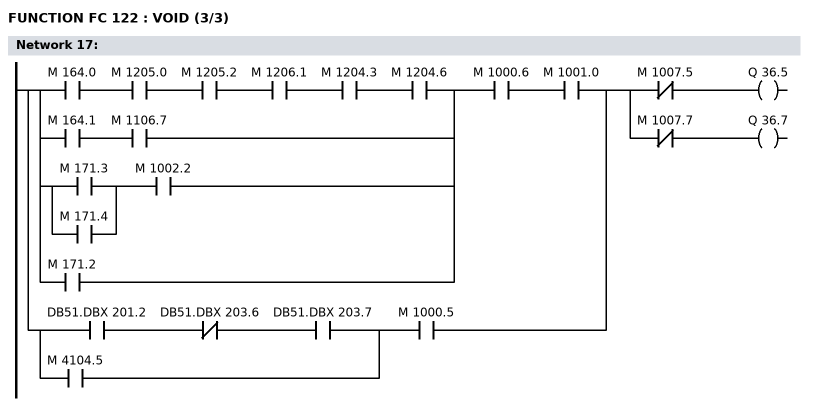

      A(    ;
      A     M    164.0;
      A     M   1205.0;
      A     M   1205.2;
      A     M   1206.1;
      A     M   1204.3;
      A     M   1204.6;
      O     ;
      A     M    164.1;
      A     M   1106.7;
      O     ;
      A(    ;
      O     M    171.3;
      O     M    171.4;
      )     ;
      A     M   1002.2;
      O     M    171.2;
      )     ;
      A     M   1000.6;
      A     M   1001.0;
      O     ;
      A(    ;
      A     DB51.DBX  201.2;
      AN    DB51.DBX  203.6;
      A     DB51.DBX  203.7;
      O     M   4104.5;
      )     ;
      A     M   1000.5;
      =     L      0.0;
      A     L      0.0;
      AN    M   1007.5;
      =     Q     36.5;
      A     L      0.0;
      AN    M   1007.7;
      =     Q     36.7;
END_FUNCTION

FUNCTION_BLOCK FB 123
TITLE =
VERSION : 0.1


VAR
  S706_LM_DC_PIN : FB 424;
  S706_LM_DC_1ST_CLAMP1 : FB 424;
  S706_LM_DC_1ST_CLAMP2 : FB 424;
  S706_LM_DC_1ST_CLAMP3 : FB 424;
  S706_LM_DC_1ST_CLAMP4 : FB 424;
  S706_LM_DC_2ND_CLAMP1 : FB 424;
  S706_LM_DC_2ND_CLAMP2 : FB 424;
  S706_LM_DC_2ND_CLAMP3 : FB 424;
  S706_LM_DC_2ND_CLAMP4 : FB 424;
  S706_LM_DC_2ND_CLAMP5 : FB 424;
  S706_LM_DC_STK_PIN : FB 424;
  S706_LM_DC_OTR_CLAMP : FB 424;
  S706_LM_DC_ASSY_CLAMP : FB 424;
  S706_LM_DC_FF_PIN : FB 424;
  S706_LM_DC_FF_CLAMP : FB 424;
  S706_LM_DC_2ND_CLAMP6 : FB 424;
  S706_LM_DC_2ND_CLAMP7 : FB 424;
  S706_LM_DC_1ST_CLAMP5 : FB 424;
END_VAR
BEGIN
NETWORK
TITLE =
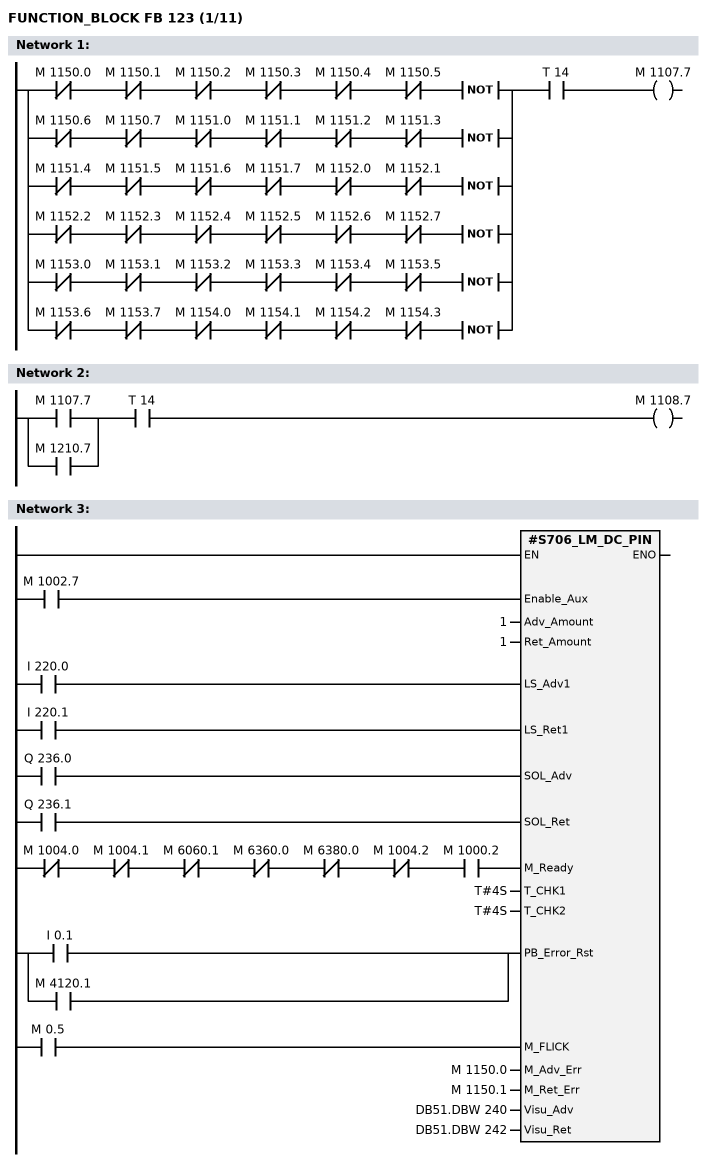

      A(    ;
      AN    M   1150.0;
      AN    M   1150.1;
      AN    M   1150.2;
      AN    M   1150.3;
      AN    M   1150.4;
      AN    M   1150.5;
      NOT   ;
      O(    ;
      AN    M   1150.6;
      AN    M   1150.7;
      AN    M   1151.0;
      AN    M   1151.1;
      AN    M   1151.2;
      AN    M   1151.3;
      NOT   ;
      )     ;
      O(    ;
      AN    M   1151.4;
      AN    M   1151.5;
      AN    M   1151.6;
      AN    M   1151.7;
      AN    M   1152.0;
      AN    M   1152.1;
      NOT   ;
      )     ;
      O(    ;
      AN    M   1152.2;
      AN    M   1152.3;
      AN    M   1152.4;
      AN    M   1152.5;
      AN    M   1152.6;
      AN    M   1152.7;
      NOT   ;
      )     ;
      O(    ;
      AN    M   1153.0;
      AN    M   1153.1;
      AN    M   1153.2;
      AN    M   1153.3;
      AN    M   1153.4;
      AN    M   1153.5;
      NOT   ;
      )     ;
      O(    ;
      AN    M   1153.6;
      AN    M   1153.7;
      AN    M   1154.0;
      AN    M   1154.1;
      AN    M   1154.2;
      AN    M   1154.3;
      NOT   ;
      )     ;
      )     ;
      A     T     14;
      =     M   1107.7;
NETWORK
TITLE =

      A(    ;
      O     M   1107.7;
      O     M   1210.7;
      )     ;
      A     T     14;
      =     M   1108.7;
NETWORK
TITLE =

      A     M   1002.7;
      =     L      0.0;
      BLD   103;
      A     I    220.0;
      =     L      0.1;
      BLD   103;
      A     I    220.1;
      =     L      0.2;
      BLD   103;
      A     Q    236.0;
      =     L      1.1;
      BLD   103;
      A     Q    236.1;
      =     L      1.2;
      BLD   103;
      AN    M   1004.0;
      AN    M   1004.1;
      AN    M   6060.1;
      AN    M   6360.0;
      AN    M   6380.0;
      AN    M   1004.2;
      A     M   1000.2;
      =     L      1.3;
      BLD   103;
      A(    ;
      O     I      0.1;
      O     M   4120.1;
      )     ;
      =     L      1.5;
      BLD   103;
      A     M      0.5;
      =     L      1.6;
      BLD   103;
      CALL #S706_LM_DC_PIN (
           Enable_Aux               := L      0.0,
           Adv_Amount               := 1,
           Ret_Amount               := 1,
           LS_Adv1                  := L      0.1,
           LS_Ret1                  := L      0.2,
           SOL_Adv                  := L      1.1,
           SOL_Ret                  := L      1.2,
           M_Ready                  := L      1.3,
           T_CHK1                   := T#4S,
           T_CHK2                   := T#4S,
           PB_Error_Rst             := L      1.5,
           M_FLICK                  := L      1.6,
           M_Adv_Err                := M   1150.0,
           M_Ret_Err                := M   1150.1,
           Visu_Adv                 := DB51.DBW  240,
           Visu_Ret                 := DB51.DBW  242);
      NOP   0;
NETWORK
TITLE =
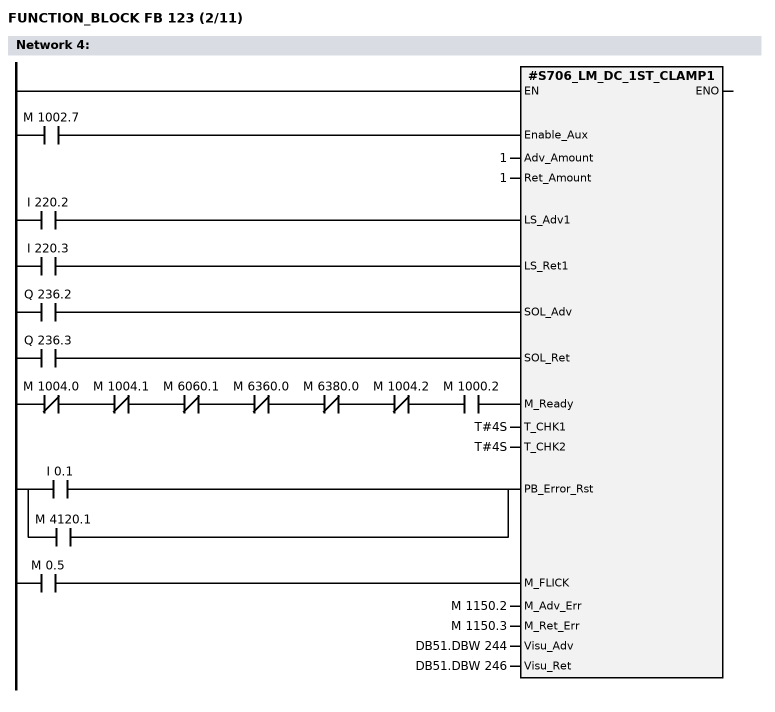

      A     M   1002.7;
      =     L      0.0;
      BLD   103;
      A     I    220.2;
      =     L      0.1;
      BLD   103;
      A     I    220.3;
      =     L      0.2;
      BLD   103;
      A     Q    236.2;
      =     L      1.1;
      BLD   103;
      A     Q    236.3;
      =     L      1.2;
      BLD   103;
      AN    M   1004.0;
      AN    M   1004.1;
      AN    M   6060.1;
      AN    M   6360.0;
      AN    M   6380.0;
      AN    M   1004.2;
      A     M   1000.2;
      =     L      1.3;
      BLD   103;
      A(    ;
      O     I      0.1;
      O     M   4120.1;
      )     ;
      =     L      1.5;
      BLD   103;
      A     M      0.5;
      =     L      1.6;
      BLD   103;
      CALL #S706_LM_DC_1ST_CLAMP1 (
           Enable_Aux               := L      0.0,
           Adv_Amount               := 1,
           Ret_Amount               := 1,
           LS_Adv1                  := L      0.1,
           LS_Ret1                  := L      0.2,
           SOL_Adv                  := L      1.1,
           SOL_Ret                  := L      1.2,
           M_Ready                  := L      1.3,
           T_CHK1                   := T#4S,
           T_CHK2                   := T#4S,
           PB_Error_Rst             := L      1.5,
           M_FLICK                  := L      1.6,
           M_Adv_Err                := M   1150.2,
           M_Ret_Err                := M   1150.3,
           Visu_Adv                 := DB51.DBW  244,
           Visu_Ret                 := DB51.DBW  246);
      NOP   0;
NETWORK
TITLE =
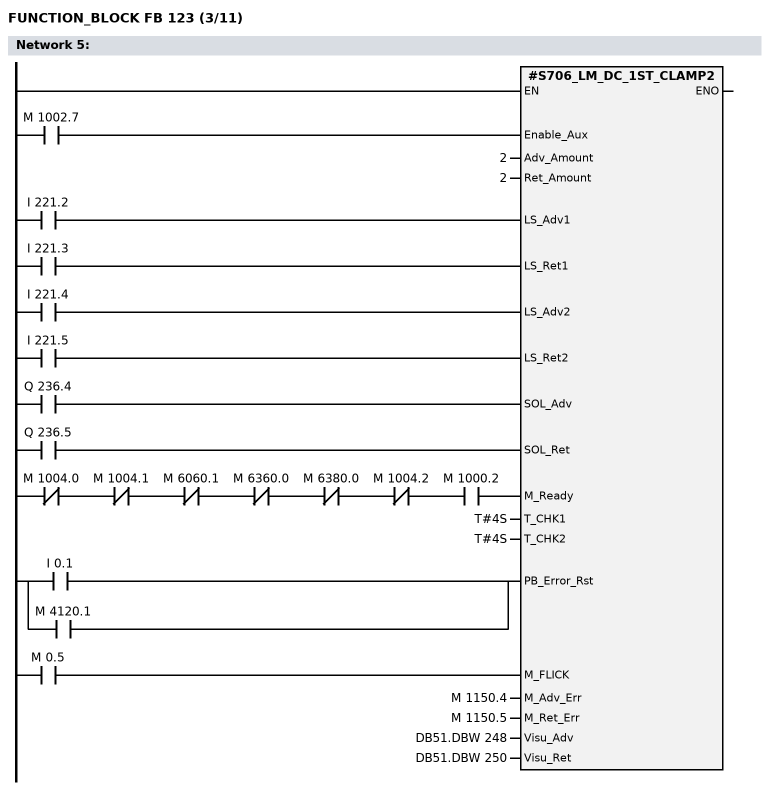

      A     M   1002.7;
      =     L      0.0;
      BLD   103;
      A     I    221.2;
      =     L      0.1;
      BLD   103;
      A     I    221.3;
      =     L      0.2;
      BLD   103;
      A     I    221.4;
      =     L      0.3;
      BLD   103;
      A     I    221.5;
      =     L      0.4;
      BLD   103;
      A     Q    236.4;
      =     L      1.1;
      BLD   103;
      A     Q    236.5;
      =     L      1.2;
      BLD   103;
      AN    M   1004.0;
      AN    M   1004.1;
      AN    M   6060.1;
      AN    M   6360.0;
      AN    M   6380.0;
      AN    M   1004.2;
      A     M   1000.2;
      =     L      1.3;
      BLD   103;
      A(    ;
      O     I      0.1;
      O     M   4120.1;
      )     ;
      =     L      1.5;
      BLD   103;
      A     M      0.5;
      =     L      1.6;
      BLD   103;
      CALL #S706_LM_DC_1ST_CLAMP2 (
           Enable_Aux               := L      0.0,
           Adv_Amount               := 2,
           Ret_Amount               := 2,
           LS_Adv1                  := L      0.1,
           LS_Ret1                  := L      0.2,
           LS_Adv2                  := L      0.3,
           LS_Ret2                  := L      0.4,
           SOL_Adv                  := L      1.1,
           SOL_Ret                  := L      1.2,
           M_Ready                  := L      1.3,
           T_CHK1                   := T#4S,
           T_CHK2                   := T#4S,
           PB_Error_Rst             := L      1.5,
           M_FLICK                  := L      1.6,
           M_Adv_Err                := M   1150.4,
           M_Ret_Err                := M   1150.5,
           Visu_Adv                 := DB51.DBW  248,
           Visu_Ret                 := DB51.DBW  250);
      NOP   0;
NETWORK
TITLE =
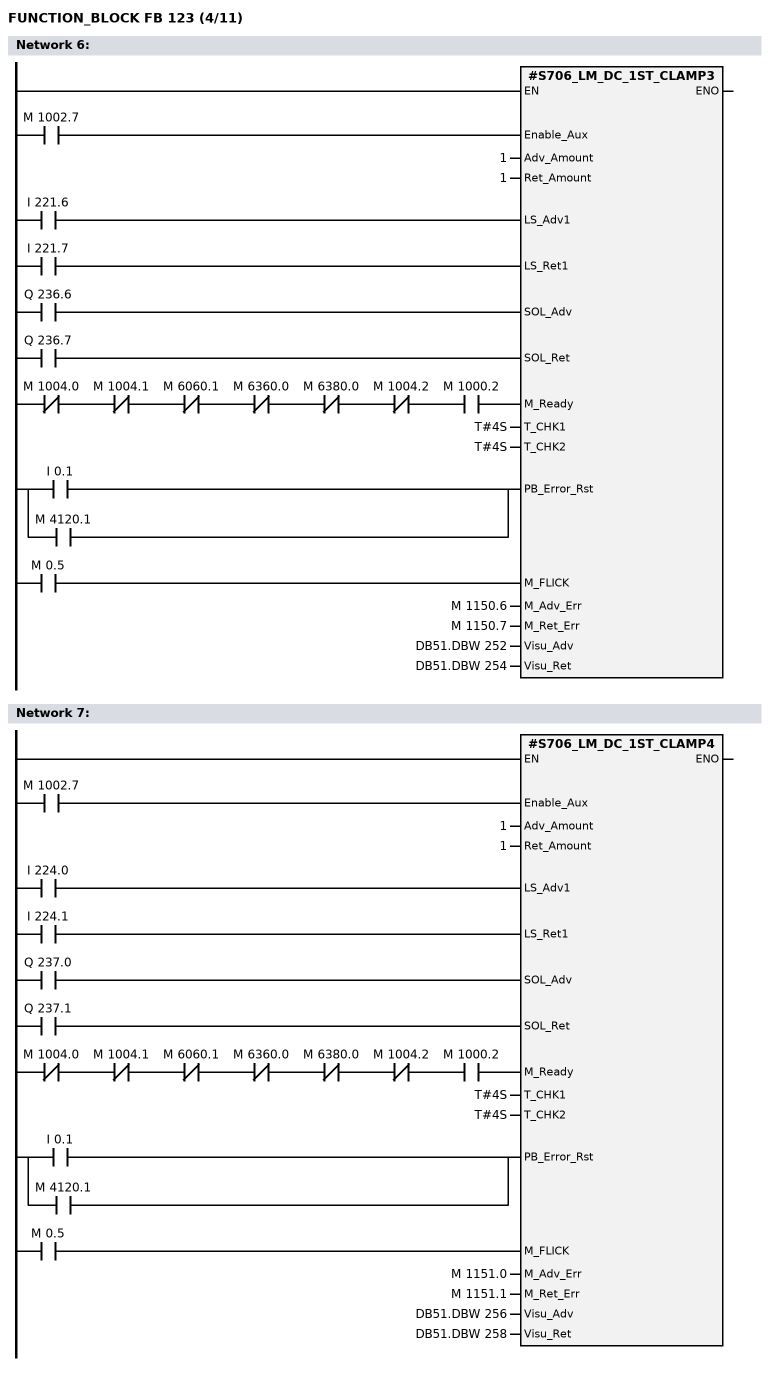

      A     M   1002.7;
      =     L      0.0;
      BLD   103;
      A     I    221.6;
      =     L      0.1;
      BLD   103;
      A     I    221.7;
      =     L      0.2;
      BLD   103;
      A     Q    236.6;
      =     L      1.1;
      BLD   103;
      A     Q    236.7;
      =     L      1.2;
      BLD   103;
      AN    M   1004.0;
      AN    M   1004.1;
      AN    M   6060.1;
      AN    M   6360.0;
      AN    M   6380.0;
      AN    M   1004.2;
      A     M   1000.2;
      =     L      1.3;
      BLD   103;
      A(    ;
      O     I      0.1;
      O     M   4120.1;
      )     ;
      =     L      1.5;
      BLD   103;
      A     M      0.5;
      =     L      1.6;
      BLD   103;
      CALL #S706_LM_DC_1ST_CLAMP3 (
           Enable_Aux               := L      0.0,
           Adv_Amount               := 1,
           Ret_Amount               := 1,
           LS_Adv1                  := L      0.1,
           LS_Ret1                  := L      0.2,
           SOL_Adv                  := L      1.1,
           SOL_Ret                  := L      1.2,
           M_Ready                  := L      1.3,
           T_CHK1                   := T#4S,
           T_CHK2                   := T#4S,
           PB_Error_Rst             := L      1.5,
           M_FLICK                  := L      1.6,
           M_Adv_Err                := M   1150.6,
           M_Ret_Err                := M   1150.7,
           Visu_Adv                 := DB51.DBW  252,
           Visu_Ret                 := DB51.DBW  254);
      NOP   0;
NETWORK
TITLE =

      A     M   1002.7;
      =     L      0.0;
      BLD   103;
      A     I    224.0;
      =     L      0.1;
      BLD   103;
      A     I    224.1;
      =     L      0.2;
      BLD   103;
      A     Q    237.0;
      =     L      1.1;
      BLD   103;
      A     Q    237.1;
      =     L      1.2;
      BLD   103;
      AN    M   1004.0;
      AN    M   1004.1;
      AN    M   6060.1;
      AN    M   6360.0;
      AN    M   6380.0;
      AN    M   1004.2;
      A     M   1000.2;
      =     L      1.3;
      BLD   103;
      A(    ;
      O     I      0.1;
      O     M   4120.1;
      )     ;
      =     L      1.5;
      BLD   103;
      A     M      0.5;
      =     L      1.6;
      BLD   103;
      CALL #S706_LM_DC_1ST_CLAMP4 (
           Enable_Aux               := L      0.0,
           Adv_Amount               := 1,
           Ret_Amount               := 1,
           LS_Adv1                  := L      0.1,
           LS_Ret1                  := L      0.2,
           SOL_Adv                  := L      1.1,
           SOL_Ret                  := L      1.2,
           M_Ready                  := L      1.3,
           T_CHK1                   := T#4S,
           T_CHK2                   := T#4S,
           PB_Error_Rst             := L      1.5,
           M_FLICK                  := L      1.6,
           M_Adv_Err                := M   1151.0,
           M_Ret_Err                := M   1151.1,
           Visu_Adv                 := DB51.DBW  256,
           Visu_Ret                 := DB51.DBW  258);
      NOP   0;
NETWORK
TITLE =
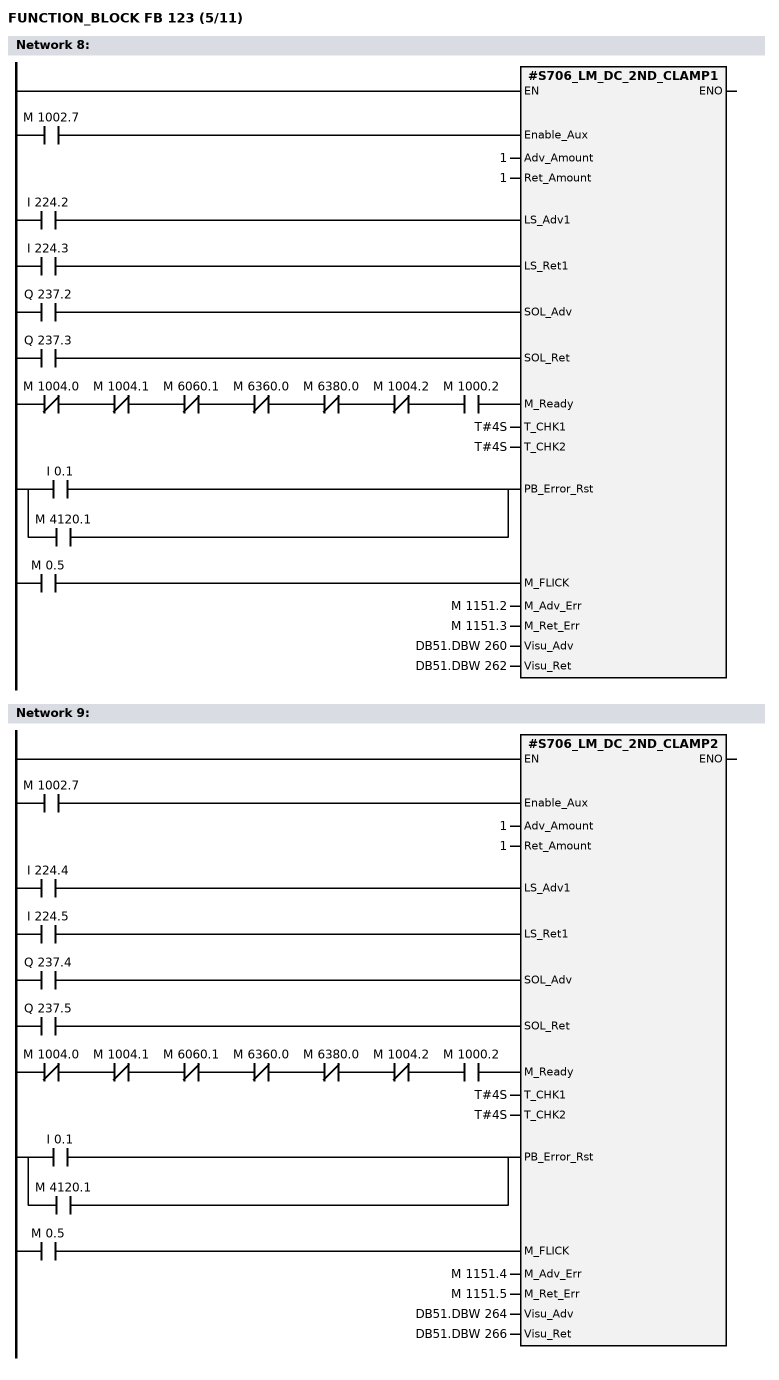

      A     M   1002.7;
      =     L      0.0;
      BLD   103;
      A     I    224.2;
      =     L      0.1;
      BLD   103;
      A     I    224.3;
      =     L      0.2;
      BLD   103;
      A     Q    237.2;
      =     L      1.1;
      BLD   103;
      A     Q    237.3;
      =     L      1.2;
      BLD   103;
      AN    M   1004.0;
      AN    M   1004.1;
      AN    M   6060.1;
      AN    M   6360.0;
      AN    M   6380.0;
      AN    M   1004.2;
      A     M   1000.2;
      =     L      1.3;
      BLD   103;
      A(    ;
      O     I      0.1;
      O     M   4120.1;
      )     ;
      =     L      1.5;
      BLD   103;
      A     M      0.5;
      =     L      1.6;
      BLD   103;
      CALL #S706_LM_DC_2ND_CLAMP1 (
           Enable_Aux               := L      0.0,
           Adv_Amount               := 1,
           Ret_Amount               := 1,
           LS_Adv1                  := L      0.1,
           LS_Ret1                  := L      0.2,
           SOL_Adv                  := L      1.1,
           SOL_Ret                  := L      1.2,
           M_Ready                  := L      1.3,
           T_CHK1                   := T#4S,
           T_CHK2                   := T#4S,
           PB_Error_Rst             := L      1.5,
           M_FLICK                  := L      1.6,
           M_Adv_Err                := M   1151.2,
           M_Ret_Err                := M   1151.3,
           Visu_Adv                 := DB51.DBW  260,
           Visu_Ret                 := DB51.DBW  262);
      NOP   0;
NETWORK
TITLE =

      A     M   1002.7;
      =     L      0.0;
      BLD   103;
      A     I    224.4;
      =     L      0.1;
      BLD   103;
      A     I    224.5;
      =     L      0.2;
      BLD   103;
      A     Q    237.4;
      =     L      1.1;
      BLD   103;
      A     Q    237.5;
      =     L      1.2;
      BLD   103;
      AN    M   1004.0;
      AN    M   1004.1;
      AN    M   6060.1;
      AN    M   6360.0;
      AN    M   6380.0;
      AN    M   1004.2;
      A     M   1000.2;
      =     L      1.3;
      BLD   103;
      A(    ;
      O     I      0.1;
      O     M   4120.1;
      )     ;
      =     L      1.5;
      BLD   103;
      A     M      0.5;
      =     L      1.6;
      BLD   103;
      CALL #S706_LM_DC_2ND_CLAMP2 (
           Enable_Aux               := L      0.0,
           Adv_Amount               := 1,
           Ret_Amount               := 1,
           LS_Adv1                  := L      0.1,
           LS_Ret1                  := L      0.2,
           SOL_Adv                  := L      1.1,
           SOL_Ret                  := L      1.2,
           M_Ready                  := L      1.3,
           T_CHK1                   := T#4S,
           T_CHK2                   := T#4S,
           PB_Error_Rst             := L      1.5,
           M_FLICK                  := L      1.6,
           M_Adv_Err                := M   1151.4,
           M_Ret_Err                := M   1151.5,
           Visu_Adv                 := DB51.DBW  264,
           Visu_Ret                 := DB51.DBW  266);
      NOP   0;
NETWORK
TITLE =
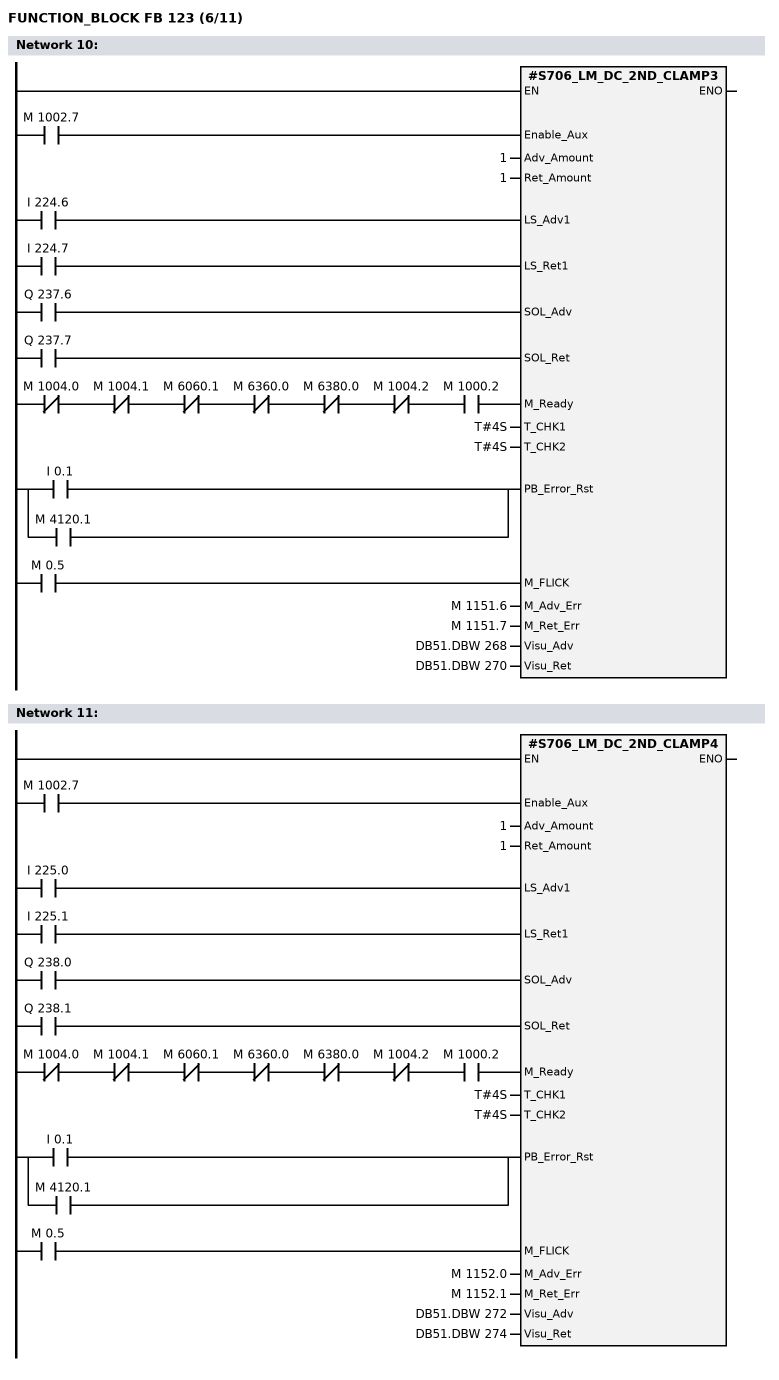

      A     M   1002.7;
      =     L      0.0;
      BLD   103;
      A     I    224.6;
      =     L      0.1;
      BLD   103;
      A     I    224.7;
      =     L      0.2;
      BLD   103;
      A     Q    237.6;
      =     L      1.1;
      BLD   103;
      A     Q    237.7;
      =     L      1.2;
      BLD   103;
      AN    M   1004.0;
      AN    M   1004.1;
      AN    M   6060.1;
      AN    M   6360.0;
      AN    M   6380.0;
      AN    M   1004.2;
      A     M   1000.2;
      =     L      1.3;
      BLD   103;
      A(    ;
      O     I      0.1;
      O     M   4120.1;
      )     ;
      =     L      1.5;
      BLD   103;
      A     M      0.5;
      =     L      1.6;
      BLD   103;
      CALL #S706_LM_DC_2ND_CLAMP3 (
           Enable_Aux               := L      0.0,
           Adv_Amount               := 1,
           Ret_Amount               := 1,
           LS_Adv1                  := L      0.1,
           LS_Ret1                  := L      0.2,
           SOL_Adv                  := L      1.1,
           SOL_Ret                  := L      1.2,
           M_Ready                  := L      1.3,
           T_CHK1                   := T#4S,
           T_CHK2                   := T#4S,
           PB_Error_Rst             := L      1.5,
           M_FLICK                  := L      1.6,
           M_Adv_Err                := M   1151.6,
           M_Ret_Err                := M   1151.7,
           Visu_Adv                 := DB51.DBW  268,
           Visu_Ret                 := DB51.DBW  270);
      NOP   0;
NETWORK
TITLE =

      A     M   1002.7;
      =     L      0.0;
      BLD   103;
      A     I    225.0;
      =     L      0.1;
      BLD   103;
      A     I    225.1;
      =     L      0.2;
      BLD   103;
      A     Q    238.0;
      =     L      1.1;
      BLD   103;
      A     Q    238.1;
      =     L      1.2;
      BLD   103;
      AN    M   1004.0;
      AN    M   1004.1;
      AN    M   6060.1;
      AN    M   6360.0;
      AN    M   6380.0;
      AN    M   1004.2;
      A     M   1000.2;
      =     L      1.3;
      BLD   103;
      A(    ;
      O     I      0.1;
      O     M   4120.1;
      )     ;
      =     L      1.5;
      BLD   103;
      A     M      0.5;
      =     L      1.6;
      BLD   103;
      CALL #S706_LM_DC_2ND_CLAMP4 (
           Enable_Aux               := L      0.0,
           Adv_Amount               := 1,
           Ret_Amount               := 1,
           LS_Adv1                  := L      0.1,
           LS_Ret1                  := L      0.2,
           SOL_Adv                  := L      1.1,
           SOL_Ret                  := L      1.2,
           M_Ready                  := L      1.3,
           T_CHK1                   := T#4S,
           T_CHK2                   := T#4S,
           PB_Error_Rst             := L      1.5,
           M_FLICK                  := L      1.6,
           M_Adv_Err                := M   1152.0,
           M_Ret_Err                := M   1152.1,
           Visu_Adv                 := DB51.DBW  272,
           Visu_Ret                 := DB51.DBW  274);
      NOP   0;
NETWORK
TITLE =
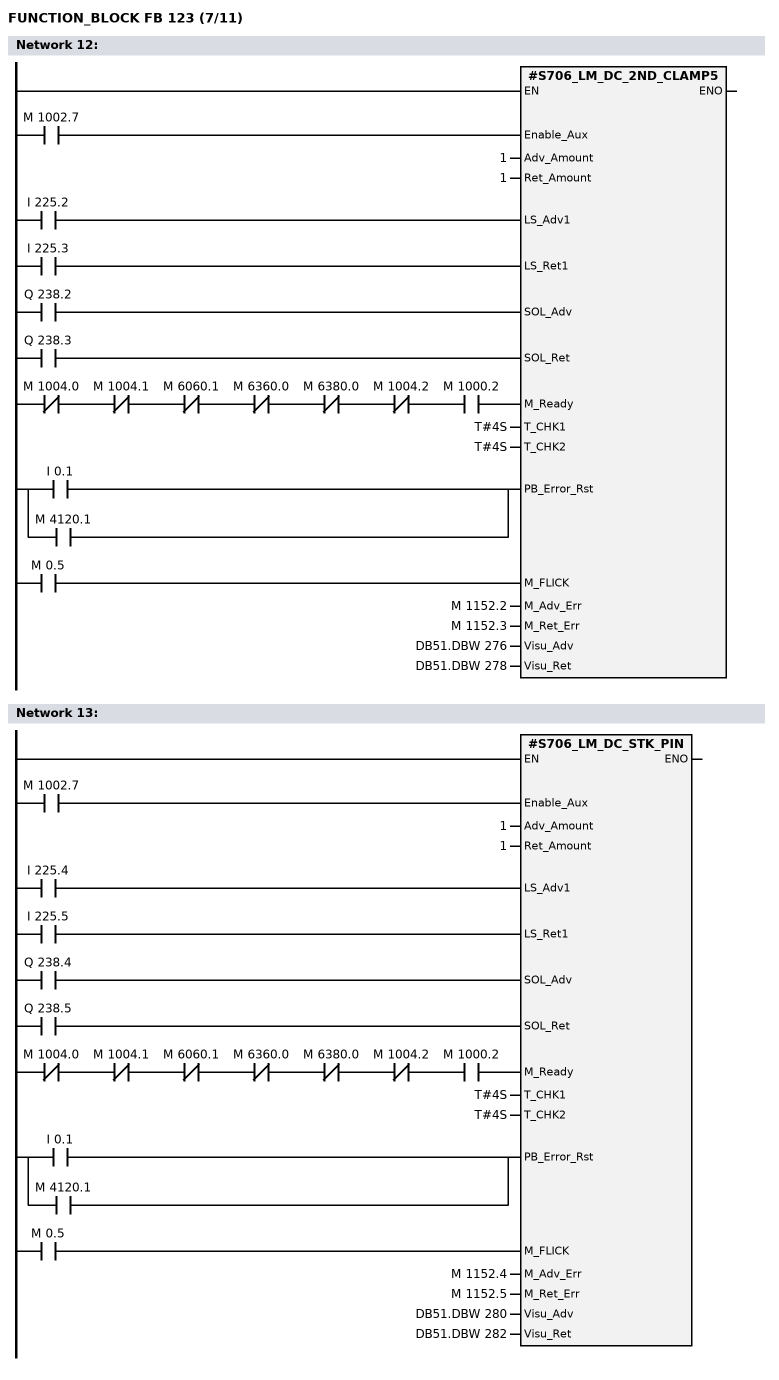

      A     M   1002.7;
      =     L      0.0;
      BLD   103;
      A     I    225.2;
      =     L      0.1;
      BLD   103;
      A     I    225.3;
      =     L      0.2;
      BLD   103;
      A     Q    238.2;
      =     L      1.1;
      BLD   103;
      A     Q    238.3;
      =     L      1.2;
      BLD   103;
      AN    M   1004.0;
      AN    M   1004.1;
      AN    M   6060.1;
      AN    M   6360.0;
      AN    M   6380.0;
      AN    M   1004.2;
      A     M   1000.2;
      =     L      1.3;
      BLD   103;
      A(    ;
      O     I      0.1;
      O     M   4120.1;
      )     ;
      =     L      1.5;
      BLD   103;
      A     M      0.5;
      =     L      1.6;
      BLD   103;
      CALL #S706_LM_DC_2ND_CLAMP5 (
           Enable_Aux               := L      0.0,
           Adv_Amount               := 1,
           Ret_Amount               := 1,
           LS_Adv1                  := L      0.1,
           LS_Ret1                  := L      0.2,
           SOL_Adv                  := L      1.1,
           SOL_Ret                  := L      1.2,
           M_Ready                  := L      1.3,
           T_CHK1                   := T#4S,
           T_CHK2                   := T#4S,
           PB_Error_Rst             := L      1.5,
           M_FLICK                  := L      1.6,
           M_Adv_Err                := M   1152.2,
           M_Ret_Err                := M   1152.3,
           Visu_Adv                 := DB51.DBW  276,
           Visu_Ret                 := DB51.DBW  278);
      NOP   0;
NETWORK
TITLE =

      A     M   1002.7;
      =     L      0.0;
      BLD   103;
      A     I    225.4;
      =     L      0.1;
      BLD   103;
      A     I    225.5;
      =     L      0.2;
      BLD   103;
      A     Q    238.4;
      =     L      1.1;
      BLD   103;
      A     Q    238.5;
      =     L      1.2;
      BLD   103;
      AN    M   1004.0;
      AN    M   1004.1;
      AN    M   6060.1;
      AN    M   6360.0;
      AN    M   6380.0;
      AN    M   1004.2;
      A     M   1000.2;
      =     L      1.3;
      BLD   103;
      A(    ;
      O     I      0.1;
      O     M   4120.1;
      )     ;
      =     L      1.5;
      BLD   103;
      A     M      0.5;
      =     L      1.6;
      BLD   103;
      CALL #S706_LM_DC_STK_PIN (
           Enable_Aux               := L      0.0,
           Adv_Amount               := 1,
           Ret_Amount               := 1,
           LS_Adv1                  := L      0.1,
           LS_Ret1                  := L      0.2,
           SOL_Adv                  := L      1.1,
           SOL_Ret                  := L      1.2,
           M_Ready                  := L      1.3,
           T_CHK1                   := T#4S,
           T_CHK2                   := T#4S,
           PB_Error_Rst             := L      1.5,
           M_FLICK                  := L      1.6,
           M_Adv_Err                := M   1152.4,
           M_Ret_Err                := M   1152.5,
           Visu_Adv                 := DB51.DBW  280,
           Visu_Ret                 := DB51.DBW  282);
      NOP   0;
NETWORK
TITLE =
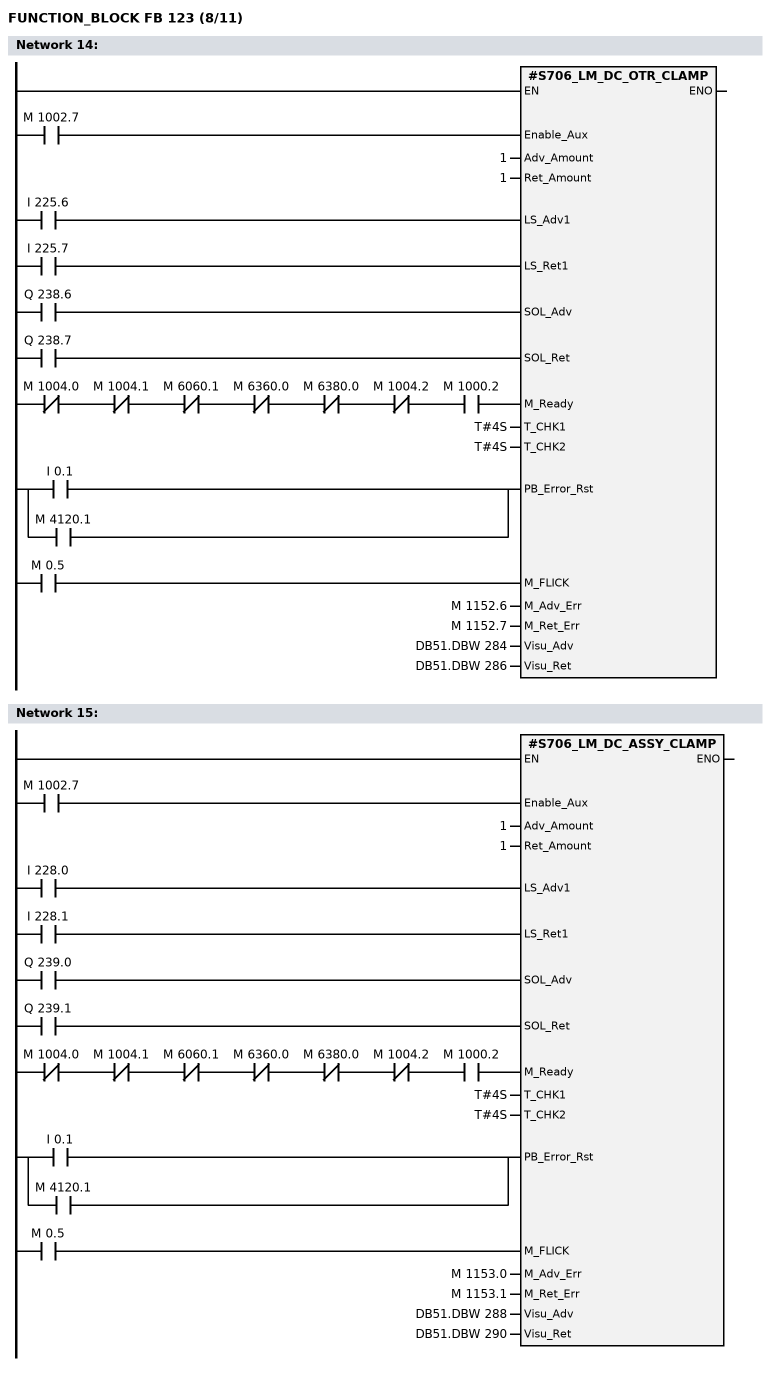

      A     M   1002.7;
      =     L      0.0;
      BLD   103;
      A     I    225.6;
      =     L      0.1;
      BLD   103;
      A     I    225.7;
      =     L      0.2;
      BLD   103;
      A     Q    238.6;
      =     L      1.1;
      BLD   103;
      A     Q    238.7;
      =     L      1.2;
      BLD   103;
      AN    M   1004.0;
      AN    M   1004.1;
      AN    M   6060.1;
      AN    M   6360.0;
      AN    M   6380.0;
      AN    M   1004.2;
      A     M   1000.2;
      =     L      1.3;
      BLD   103;
      A(    ;
      O     I      0.1;
      O     M   4120.1;
      )     ;
      =     L      1.5;
      BLD   103;
      A     M      0.5;
      =     L      1.6;
      BLD   103;
      CALL #S706_LM_DC_OTR_CLAMP (
           Enable_Aux               := L      0.0,
           Adv_Amount               := 1,
           Ret_Amount               := 1,
           LS_Adv1                  := L      0.1,
           LS_Ret1                  := L      0.2,
           SOL_Adv                  := L      1.1,
           SOL_Ret                  := L      1.2,
           M_Ready                  := L      1.3,
           T_CHK1                   := T#4S,
           T_CHK2                   := T#4S,
           PB_Error_Rst             := L      1.5,
           M_FLICK                  := L      1.6,
           M_Adv_Err                := M   1152.6,
           M_Ret_Err                := M   1152.7,
           Visu_Adv                 := DB51.DBW  284,
           Visu_Ret                 := DB51.DBW  286);
      NOP   0;
NETWORK
TITLE =

      A     M   1002.7;
      =     L      0.0;
      BLD   103;
      A     I    228.0;
      =     L      0.1;
      BLD   103;
      A     I    228.1;
      =     L      0.2;
      BLD   103;
      A     Q    239.0;
      =     L      1.1;
      BLD   103;
      A     Q    239.1;
      =     L      1.2;
      BLD   103;
      AN    M   1004.0;
      AN    M   1004.1;
      AN    M   6060.1;
      AN    M   6360.0;
      AN    M   6380.0;
      AN    M   1004.2;
      A     M   1000.2;
      =     L      1.3;
      BLD   103;
      A(    ;
      O     I      0.1;
      O     M   4120.1;
      )     ;
      =     L      1.5;
      BLD   103;
      A     M      0.5;
      =     L      1.6;
      BLD   103;
      CALL #S706_LM_DC_ASSY_CLAMP (
           Enable_Aux               := L      0.0,
           Adv_Amount               := 1,
           Ret_Amount               := 1,
           LS_Adv1                  := L      0.1,
           LS_Ret1                  := L      0.2,
           SOL_Adv                  := L      1.1,
           SOL_Ret                  := L      1.2,
           M_Ready                  := L      1.3,
           T_CHK1                   := T#4S,
           T_CHK2                   := T#4S,
           PB_Error_Rst             := L      1.5,
           M_FLICK                  := L      1.6,
           M_Adv_Err                := M   1153.0,
           M_Ret_Err                := M   1153.1,
           Visu_Adv                 := DB51.DBW  288,
           Visu_Ret                 := DB51.DBW  290);
      NOP   0;
NETWORK
TITLE =
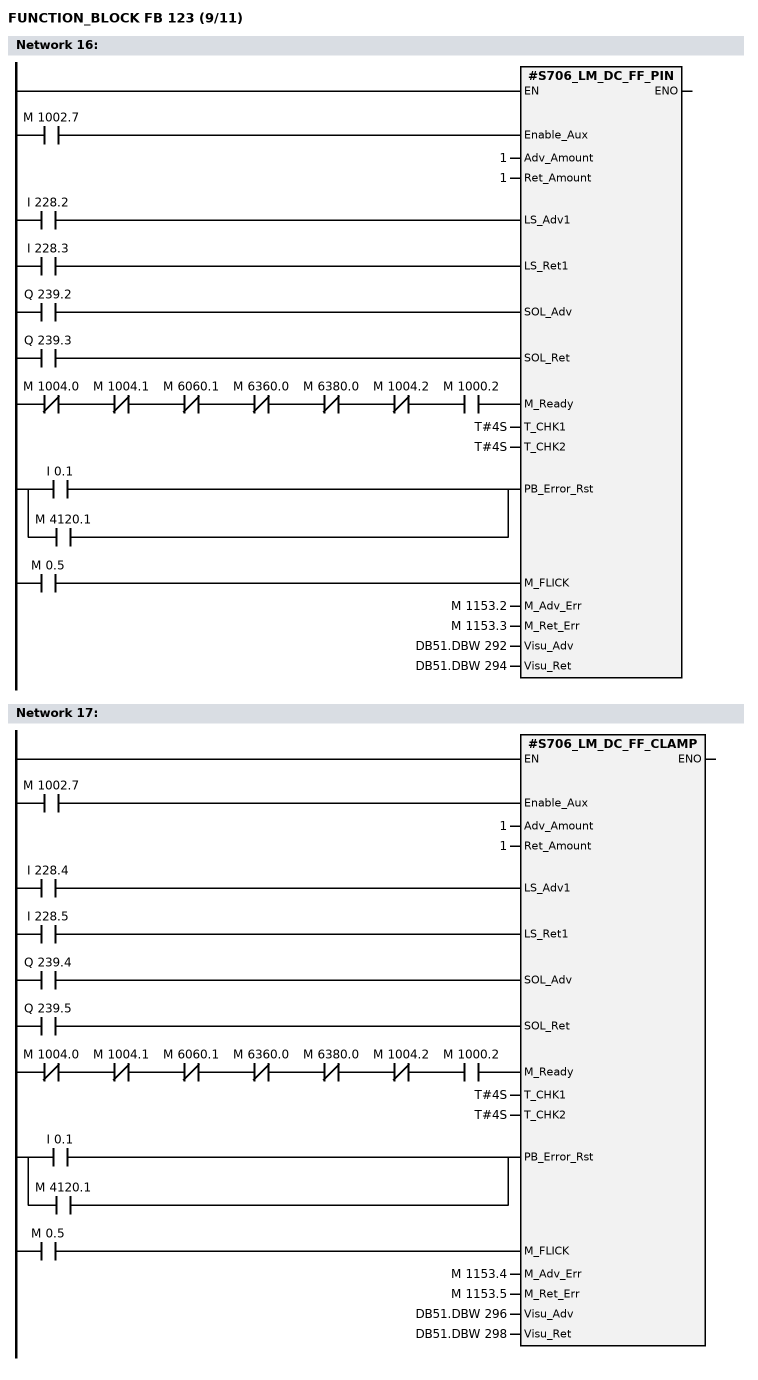

      A     M   1002.7;
      =     L      0.0;
      BLD   103;
      A     I    228.2;
      =     L      0.1;
      BLD   103;
      A     I    228.3;
      =     L      0.2;
      BLD   103;
      A     Q    239.2;
      =     L      1.1;
      BLD   103;
      A     Q    239.3;
      =     L      1.2;
      BLD   103;
      AN    M   1004.0;
      AN    M   1004.1;
      AN    M   6060.1;
      AN    M   6360.0;
      AN    M   6380.0;
      AN    M   1004.2;
      A     M   1000.2;
      =     L      1.3;
      BLD   103;
      A(    ;
      O     I      0.1;
      O     M   4120.1;
      )     ;
      =     L      1.5;
      BLD   103;
      A     M      0.5;
      =     L      1.6;
      BLD   103;
      CALL #S706_LM_DC_FF_PIN (
           Enable_Aux               := L      0.0,
           Adv_Amount               := 1,
           Ret_Amount               := 1,
           LS_Adv1                  := L      0.1,
           LS_Ret1                  := L      0.2,
           SOL_Adv                  := L      1.1,
           SOL_Ret                  := L      1.2,
           M_Ready                  := L      1.3,
           T_CHK1                   := T#4S,
           T_CHK2                   := T#4S,
           PB_Error_Rst             := L      1.5,
           M_FLICK                  := L      1.6,
           M_Adv_Err                := M   1153.2,
           M_Ret_Err                := M   1153.3,
           Visu_Adv                 := DB51.DBW  292,
           Visu_Ret                 := DB51.DBW  294);
      NOP   0;
NETWORK
TITLE =

      A     M   1002.7;
      =     L      0.0;
      BLD   103;
      A     I    228.4;
      =     L      0.1;
      BLD   103;
      A     I    228.5;
      =     L      0.2;
      BLD   103;
      A     Q    239.4;
      =     L      1.1;
      BLD   103;
      A     Q    239.5;
      =     L      1.2;
      BLD   103;
      AN    M   1004.0;
      AN    M   1004.1;
      AN    M   6060.1;
      AN    M   6360.0;
      AN    M   6380.0;
      AN    M   1004.2;
      A     M   1000.2;
      =     L      1.3;
      BLD   103;
      A(    ;
      O     I      0.1;
      O     M   4120.1;
      )     ;
      =     L      1.5;
      BLD   103;
      A     M      0.5;
      =     L      1.6;
      BLD   103;
      CALL #S706_LM_DC_FF_CLAMP (
           Enable_Aux               := L      0.0,
           Adv_Amount               := 1,
           Ret_Amount               := 1,
           LS_Adv1                  := L      0.1,
           LS_Ret1                  := L      0.2,
           SOL_Adv                  := L      1.1,
           SOL_Ret                  := L      1.2,
           M_Ready                  := L      1.3,
           T_CHK1                   := T#4S,
           T_CHK2                   := T#4S,
           PB_Error_Rst             := L      1.5,
           M_FLICK                  := L      1.6,
           M_Adv_Err                := M   1153.4,
           M_Ret_Err                := M   1153.5,
           Visu_Adv                 := DB51.DBW  296,
           Visu_Ret                 := DB51.DBW  298);
      NOP   0;
NETWORK
TITLE =
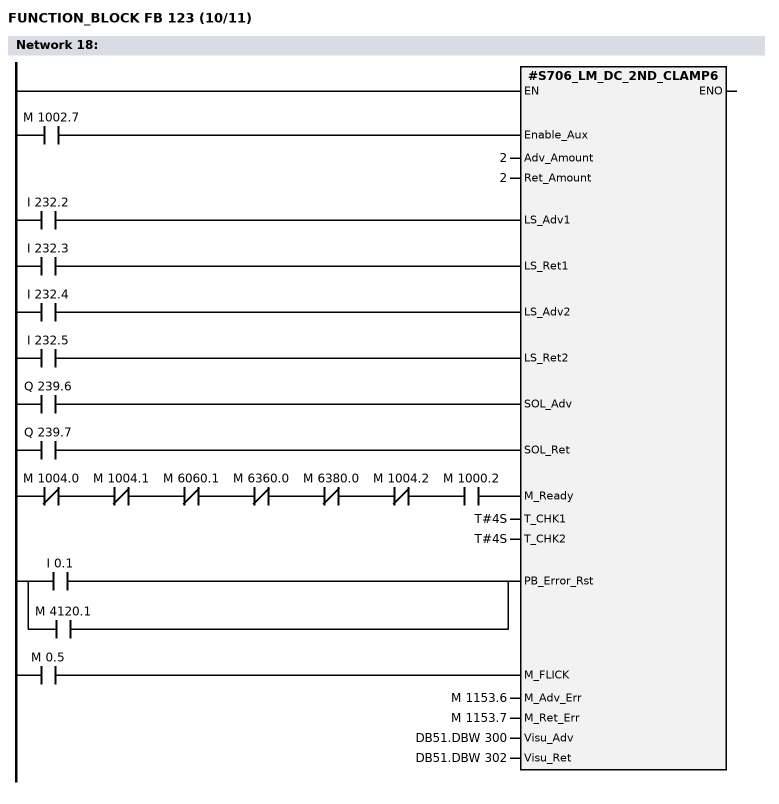

      A     M   1002.7;
      =     L      0.0;
      BLD   103;
      A     I    232.2;
      =     L      0.1;
      BLD   103;
      A     I    232.3;
      =     L      0.2;
      BLD   103;
      A     I    232.4;
      =     L      0.3;
      BLD   103;
      A     I    232.5;
      =     L      0.4;
      BLD   103;
      A     Q    239.6;
      =     L      1.1;
      BLD   103;
      A     Q    239.7;
      =     L      1.2;
      BLD   103;
      AN    M   1004.0;
      AN    M   1004.1;
      AN    M   6060.1;
      AN    M   6360.0;
      AN    M   6380.0;
      AN    M   1004.2;
      A     M   1000.2;
      =     L      1.3;
      BLD   103;
      A(    ;
      O     I      0.1;
      O     M   4120.1;
      )     ;
      =     L      1.5;
      BLD   103;
      A     M      0.5;
      =     L      1.6;
      BLD   103;
      CALL #S706_LM_DC_2ND_CLAMP6 (
           Enable_Aux               := L      0.0,
           Adv_Amount               := 2,
           Ret_Amount               := 2,
           LS_Adv1                  := L      0.1,
           LS_Ret1                  := L      0.2,
           LS_Adv2                  := L      0.3,
           LS_Ret2                  := L      0.4,
           SOL_Adv                  := L      1.1,
           SOL_Ret                  := L      1.2,
           M_Ready                  := L      1.3,
           T_CHK1                   := T#4S,
           T_CHK2                   := T#4S,
           PB_Error_Rst             := L      1.5,
           M_FLICK                  := L      1.6,
           M_Adv_Err                := M   1153.6,
           M_Ret_Err                := M   1153.7,
           Visu_Adv                 := DB51.DBW  300,
           Visu_Ret                 := DB51.DBW  302);
      NOP   0;
NETWORK
TITLE =
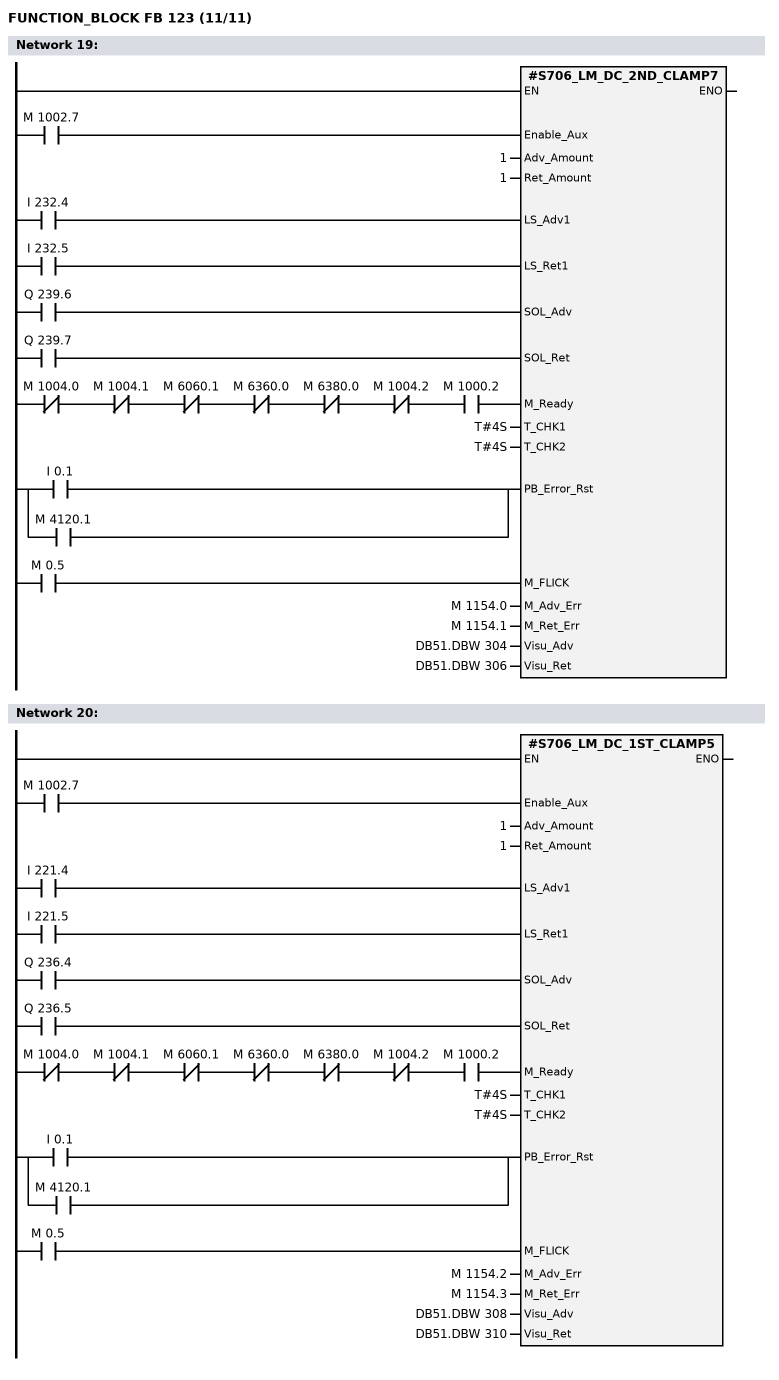

      A     M   1002.7;
      =     L      0.0;
      BLD   103;
      A     I    232.4;
      =     L      0.1;
      BLD   103;
      A     I    232.5;
      =     L      0.2;
      BLD   103;
      A     Q    239.6;
      =     L      1.1;
      BLD   103;
      A     Q    239.7;
      =     L      1.2;
      BLD   103;
      AN    M   1004.0;
      AN    M   1004.1;
      AN    M   6060.1;
      AN    M   6360.0;
      AN    M   6380.0;
      AN    M   1004.2;
      A     M   1000.2;
      =     L      1.3;
      BLD   103;
      A(    ;
      O     I      0.1;
      O     M   4120.1;
      )     ;
      =     L      1.5;
      BLD   103;
      A     M      0.5;
      =     L      1.6;
      BLD   103;
      CALL #S706_LM_DC_2ND_CLAMP7 (
           Enable_Aux               := L      0.0,
           Adv_Amount               := 1,
           Ret_Amount               := 1,
           LS_Adv1                  := L      0.1,
           LS_Ret1                  := L      0.2,
           SOL_Adv                  := L      1.1,
           SOL_Ret                  := L      1.2,
           M_Ready                  := L      1.3,
           T_CHK1                   := T#4S,
           T_CHK2                   := T#4S,
           PB_Error_Rst             := L      1.5,
           M_FLICK                  := L      1.6,
           M_Adv_Err                := M   1154.0,
           M_Ret_Err                := M   1154.1,
           Visu_Adv                 := DB51.DBW  304,
           Visu_Ret                 := DB51.DBW  306);
      NOP   0;
NETWORK
TITLE =

      A     M   1002.7;
      =     L      0.0;
      BLD   103;
      A     I    221.4;
      =     L      0.1;
      BLD   103;
      A     I    221.5;
      =     L      0.2;
      BLD   103;
      A     Q    236.4;
      =     L      1.1;
      BLD   103;
      A     Q    236.5;
      =     L      1.2;
      BLD   103;
      AN    M   1004.0;
      AN    M   1004.1;
      AN    M   6060.1;
      AN    M   6360.0;
      AN    M   6380.0;
      AN    M   1004.2;
      A     M   1000.2;
      =     L      1.3;
      BLD   103;
      A(    ;
      O     I      0.1;
      O     M   4120.1;
      )     ;
      =     L      1.5;
      BLD   103;
      A     M      0.5;
      =     L      1.6;
      BLD   103;
      CALL #S706_LM_DC_1ST_CLAMP5 (
           Enable_Aux               := L      0.0,
           Adv_Amount               := 1,
           Ret_Amount               := 1,
           LS_Adv1                  := L      0.1,
           LS_Ret1                  := L      0.2,
           SOL_Adv                  := L      1.1,
           SOL_Ret                  := L      1.2,
           M_Ready                  := L      1.3,
           T_CHK1                   := T#4S,
           T_CHK2                   := T#4S,
           PB_Error_Rst             := L      1.5,
           M_FLICK                  := L      1.6,
           M_Adv_Err                := M   1154.2,
           M_Ret_Err                := M   1154.3,
           Visu_Adv                 := DB51.DBW  308,
           Visu_Ret                 := DB51.DBW  310);
      NOP   0;
END_FUNCTION_BLOCK

DATA_BLOCK DB 123
TITLE =
VERSION : 0.0

 FB 123
BEGIN
   S706_LM_DC_PIN.Enable_Aux := FALSE;
   S706_LM_DC_PIN.Adv_Amount := 1;
   S706_LM_DC_PIN.Ret_Amount := 1;
   S706_LM_DC_PIN.LS_Adv1 := FALSE;
   S706_LM_DC_PIN.LS_Ret1 := FALSE;
   S706_LM_DC_PIN.LS_Adv2 := FALSE;
   S706_LM_DC_PIN.LS_Ret2 := FALSE;
   S706_LM_DC_PIN.LS_Adv3 := FALSE;
   S706_LM_DC_PIN.LS_Ret3 := FALSE;
   S706_LM_DC_PIN.LS_Adv4 := FALSE;
   S706_LM_DC_PIN.LS_Ret4 := FALSE;
   S706_LM_DC_PIN.SOL_Adv := FALSE;
   S706_LM_DC_PIN.SOL_Ret := FALSE;
   S706_LM_DC_PIN.M_Ready := TRUE;
   S706_LM_DC_PIN.T_CHK1 := T#4S;
   S706_LM_DC_PIN.T_CHK2 := T#4S;
   S706_LM_DC_PIN.PB_Lamp_CHK := FALSE;
   S706_LM_DC_PIN.PB_Error_Rst := FALSE;
   S706_LM_DC_PIN.M_FLICK := FALSE;
   S706_LM_DC_PIN.M_Adv_Err := FALSE;
   S706_LM_DC_PIN.M_Ret_Err := FALSE;
   S706_LM_DC_PIN.LP_Adv := FALSE;
   S706_LM_DC_PIN.LP_Ret := FALSE;
   S706_LM_DC_PIN.Visu_Adv := W#16#0;
   S706_LM_DC_PIN.Visu_Ret := W#16#0;
   S706_LM_DC_PIN.Error_T1.IN := FALSE;
   S706_LM_DC_PIN.Error_T1.PT := T#4S;
   S706_LM_DC_PIN.Error_T1.Q := FALSE;
   S706_LM_DC_PIN.Error_T1.ET := T#0MS;
   S706_LM_DC_PIN.Error_T1.STATE := B#16#0;
   S706_LM_DC_PIN.Error_T1.STIME := T#0MS;
   S706_LM_DC_PIN.Error_T1.ATIME := T#0MS;
   S706_LM_DC_PIN.Error_T2.IN := FALSE;
   S706_LM_DC_PIN.Error_T2.PT := T#4S;
   S706_LM_DC_PIN.Error_T2.Q := FALSE;
   S706_LM_DC_PIN.Error_T2.ET := T#0MS;
   S706_LM_DC_PIN.Error_T2.STATE := B#16#0;
   S706_LM_DC_PIN.Error_T2.STIME := T#0MS;
   S706_LM_DC_PIN.Error_T2.ATIME := T#0MS;
   S706_LM_DC_PIN.CHK_Aux1 := FALSE;
   S706_LM_DC_PIN.CHK_Aux2 := FALSE;
   S706_LM_DC_PIN.Error_T1_DN := FALSE;
   S706_LM_DC_PIN.Error_T2_DN := FALSE;
   S706_LM_DC_PIN.Adv_Memo := TRUE;
   S706_LM_DC_PIN.Visu_Adv_Arr[0] := FALSE;
   S706_LM_DC_PIN.Visu_Adv_Arr[1] := FALSE;
   S706_LM_DC_PIN.Visu_Adv_Arr[2] := FALSE;
   S706_LM_DC_PIN.Visu_Adv_Arr[3] := FALSE;
   S706_LM_DC_PIN.Visu_Adv_Arr[4] := FALSE;
   S706_LM_DC_PIN.Visu_Adv_Arr[5] := FALSE;
   S706_LM_DC_PIN.Visu_Adv_Arr[6] := FALSE;
   S706_LM_DC_PIN.Visu_Adv_Arr[7] := FALSE;
   S706_LM_DC_PIN.Visu_Adv_Arr[8] := FALSE;
   S706_LM_DC_PIN.Visu_Adv_Arr[9] := FALSE;
   S706_LM_DC_PIN.Visu_Adv_Arr[10] := FALSE;
   S706_LM_DC_PIN.Visu_Adv_Arr[11] := FALSE;
   S706_LM_DC_PIN.Visu_Adv_Arr[12] := FALSE;
   S706_LM_DC_PIN.Visu_Adv_Arr[13] := FALSE;
   S706_LM_DC_PIN.Visu_Adv_Arr[14] := FALSE;
   S706_LM_DC_PIN.Visu_Adv_Arr[15] := FALSE;
   S706_LM_DC_PIN.Visu_Ret_Arr[0] := FALSE;
   S706_LM_DC_PIN.Visu_Ret_Arr[1] := FALSE;
   S706_LM_DC_PIN.Visu_Ret_Arr[2] := FALSE;
   S706_LM_DC_PIN.Visu_Ret_Arr[3] := FALSE;
   S706_LM_DC_PIN.Visu_Ret_Arr[4] := FALSE;
   S706_LM_DC_PIN.Visu_Ret_Arr[5] := FALSE;
   S706_LM_DC_PIN.Visu_Ret_Arr[6] := FALSE;
   S706_LM_DC_PIN.Visu_Ret_Arr[7] := FALSE;
   S706_LM_DC_PIN.Visu_Ret_Arr[8] := FALSE;
   S706_LM_DC_PIN.Visu_Ret_Arr[9] := FALSE;
   S706_LM_DC_PIN.Visu_Ret_Arr[10] := FALSE;
   S706_LM_DC_PIN.Visu_Ret_Arr[11] := FALSE;
   S706_LM_DC_PIN.Visu_Ret_Arr[12] := FALSE;
   S706_LM_DC_PIN.Visu_Ret_Arr[13] := FALSE;
   S706_LM_DC_PIN.Visu_Ret_Arr[14] := FALSE;
   S706_LM_DC_PIN.Visu_Ret_Arr[15] := FALSE;
   S706_LM_DC_PIN.BLK_Move_Ret := 0;
   S706_LM_DC_PIN.Enable := FALSE;
   S706_LM_DC_PIN.Adv_End := FALSE;
   S706_LM_DC_PIN.Ret_End := FALSE;
   S706_LM_DC_1ST_CLAMP1.Enable_Aux := FALSE;
   S706_LM_DC_1ST_CLAMP1.Adv_Amount := 1;
   S706_LM_DC_1ST_CLAMP1.Ret_Amount := 1;
   S706_LM_DC_1ST_CLAMP1.LS_Adv1 := FALSE;
   S706_LM_DC_1ST_CLAMP1.LS_Ret1 := FALSE;
   S706_LM_DC_1ST_CLAMP1.LS_Adv2 := FALSE;
   S706_LM_DC_1ST_CLAMP1.LS_Ret2 := FALSE;
   S706_LM_DC_1ST_CLAMP1.LS_Adv3 := FALSE;
   S706_LM_DC_1ST_CLAMP1.LS_Ret3 := FALSE;
   S706_LM_DC_1ST_CLAMP1.LS_Adv4 := FALSE;
   S706_LM_DC_1ST_CLAMP1.LS_Ret4 := FALSE;
   S706_LM_DC_1ST_CLAMP1.SOL_Adv := FALSE;
   S706_LM_DC_1ST_CLAMP1.SOL_Ret := FALSE;
   S706_LM_DC_1ST_CLAMP1.M_Ready := TRUE;
   S706_LM_DC_1ST_CLAMP1.T_CHK1 := T#4S;
   S706_LM_DC_1ST_CLAMP1.T_CHK2 := T#4S;
   S706_LM_DC_1ST_CLAMP1.PB_Lamp_CHK := FALSE;
   S706_LM_DC_1ST_CLAMP1.PB_Error_Rst := FALSE;
   S706_LM_DC_1ST_CLAMP1.M_FLICK := FALSE;
   S706_LM_DC_1ST_CLAMP1.M_Adv_Err := FALSE;
   S706_LM_DC_1ST_CLAMP1.M_Ret_Err := FALSE;
   S706_LM_DC_1ST_CLAMP1.LP_Adv := FALSE;
   S706_LM_DC_1ST_CLAMP1.LP_Ret := FALSE;
   S706_LM_DC_1ST_CLAMP1.Visu_Adv := W#16#0;
   S706_LM_DC_1ST_CLAMP1.Visu_Ret := W#16#0;
   S706_LM_DC_1ST_CLAMP1.Error_T1.IN := FALSE;
   S706_LM_DC_1ST_CLAMP1.Error_T1.PT := T#4S;
   S706_LM_DC_1ST_CLAMP1.Error_T1.Q := FALSE;
   S706_LM_DC_1ST_CLAMP1.Error_T1.ET := T#0MS;
   S706_LM_DC_1ST_CLAMP1.Error_T1.STATE := B#16#0;
   S706_LM_DC_1ST_CLAMP1.Error_T1.STIME := T#0MS;
   S706_LM_DC_1ST_CLAMP1.Error_T1.ATIME := T#0MS;
   S706_LM_DC_1ST_CLAMP1.Error_T2.IN := FALSE;
   S706_LM_DC_1ST_CLAMP1.Error_T2.PT := T#4S;
   S706_LM_DC_1ST_CLAMP1.Error_T2.Q := FALSE;
   S706_LM_DC_1ST_CLAMP1.Error_T2.ET := T#0MS;
   S706_LM_DC_1ST_CLAMP1.Error_T2.STATE := B#16#0;
   S706_LM_DC_1ST_CLAMP1.Error_T2.STIME := T#0MS;
   S706_LM_DC_1ST_CLAMP1.Error_T2.ATIME := T#0MS;
   S706_LM_DC_1ST_CLAMP1.CHK_Aux1 := FALSE;
   S706_LM_DC_1ST_CLAMP1.CHK_Aux2 := FALSE;
   S706_LM_DC_1ST_CLAMP1.Error_T1_DN := FALSE;
   S706_LM_DC_1ST_CLAMP1.Error_T2_DN := FALSE;
   S706_LM_DC_1ST_CLAMP1.Adv_Memo := TRUE;
   S706_LM_DC_1ST_CLAMP1.Visu_Adv_Arr[0] := FALSE;
   S706_LM_DC_1ST_CLAMP1.Visu_Adv_Arr[1] := FALSE;
   S706_LM_DC_1ST_CLAMP1.Visu_Adv_Arr[2] := FALSE;
   S706_LM_DC_1ST_CLAMP1.Visu_Adv_Arr[3] := FALSE;
   S706_LM_DC_1ST_CLAMP1.Visu_Adv_Arr[4] := FALSE;
   S706_LM_DC_1ST_CLAMP1.Visu_Adv_Arr[5] := FALSE;
   S706_LM_DC_1ST_CLAMP1.Visu_Adv_Arr[6] := FALSE;
   S706_LM_DC_1ST_CLAMP1.Visu_Adv_Arr[7] := FALSE;
   S706_LM_DC_1ST_CLAMP1.Visu_Adv_Arr[8] := FALSE;
   S706_LM_DC_1ST_CLAMP1.Visu_Adv_Arr[9] := FALSE;
   S706_LM_DC_1ST_CLAMP1.Visu_Adv_Arr[10] := FALSE;
   S706_LM_DC_1ST_CLAMP1.Visu_Adv_Arr[11] := FALSE;
   S706_LM_DC_1ST_CLAMP1.Visu_Adv_Arr[12] := FALSE;
   S706_LM_DC_1ST_CLAMP1.Visu_Adv_Arr[13] := FALSE;
   S706_LM_DC_1ST_CLAMP1.Visu_Adv_Arr[14] := FALSE;
   S706_LM_DC_1ST_CLAMP1.Visu_Adv_Arr[15] := FALSE;
   S706_LM_DC_1ST_CLAMP1.Visu_Ret_Arr[0] := FALSE;
   S706_LM_DC_1ST_CLAMP1.Visu_Ret_Arr[1] := FALSE;
   S706_LM_DC_1ST_CLAMP1.Visu_Ret_Arr[2] := FALSE;
   S706_LM_DC_1ST_CLAMP1.Visu_Ret_Arr[3] := FALSE;
   S706_LM_DC_1ST_CLAMP1.Visu_Ret_Arr[4] := FALSE;
   S706_LM_DC_1ST_CLAMP1.Visu_Ret_Arr[5] := FALSE;
   S706_LM_DC_1ST_CLAMP1.Visu_Ret_Arr[6] := FALSE;
   S706_LM_DC_1ST_CLAMP1.Visu_Ret_Arr[7] := FALSE;
   S706_LM_DC_1ST_CLAMP1.Visu_Ret_Arr[8] := FALSE;
   S706_LM_DC_1ST_CLAMP1.Visu_Ret_Arr[9] := FALSE;
   S706_LM_DC_1ST_CLAMP1.Visu_Ret_Arr[10] := FALSE;
   S706_LM_DC_1ST_CLAMP1.Visu_Ret_Arr[11] := FALSE;
   S706_LM_DC_1ST_CLAMP1.Visu_Ret_Arr[12] := FALSE;
   S706_LM_DC_1ST_CLAMP1.Visu_Ret_Arr[13] := FALSE;
   S706_LM_DC_1ST_CLAMP1.Visu_Ret_Arr[14] := FALSE;
   S706_LM_DC_1ST_CLAMP1.Visu_Ret_Arr[15] := FALSE;
   S706_LM_DC_1ST_CLAMP1.BLK_Move_Ret := 0;
   S706_LM_DC_1ST_CLAMP1.Enable := FALSE;
   S706_LM_DC_1ST_CLAMP1.Adv_End := FALSE;
   S706_LM_DC_1ST_CLAMP1.Ret_End := FALSE;
   S706_LM_DC_1ST_CLAMP2.Enable_Aux := FALSE;
   S706_LM_DC_1ST_CLAMP2.Adv_Amount := 2;
   S706_LM_DC_1ST_CLAMP2.Ret_Amount := 2;
   S706_LM_DC_1ST_CLAMP2.LS_Adv1 := FALSE;
   S706_LM_DC_1ST_CLAMP2.LS_Ret1 := FALSE;
   S706_LM_DC_1ST_CLAMP2.LS_Adv2 := FALSE;
   S706_LM_DC_1ST_CLAMP2.LS_Ret2 := FALSE;
   S706_LM_DC_1ST_CLAMP2.LS_Adv3 := FALSE;
   S706_LM_DC_1ST_CLAMP2.LS_Ret3 := FALSE;
   S706_LM_DC_1ST_CLAMP2.LS_Adv4 := FALSE;
   S706_LM_DC_1ST_CLAMP2.LS_Ret4 := FALSE;
   S706_LM_DC_1ST_CLAMP2.SOL_Adv := FALSE;
   S706_LM_DC_1ST_CLAMP2.SOL_Ret := FALSE;
   S706_LM_DC_1ST_CLAMP2.M_Ready := TRUE;
   S706_LM_DC_1ST_CLAMP2.T_CHK1 := T#4S;
   S706_LM_DC_1ST_CLAMP2.T_CHK2 := T#4S;
   S706_LM_DC_1ST_CLAMP2.PB_Lamp_CHK := FALSE;
   S706_LM_DC_1ST_CLAMP2.PB_Error_Rst := FALSE;
   S706_LM_DC_1ST_CLAMP2.M_FLICK := FALSE;
   S706_LM_DC_1ST_CLAMP2.M_Adv_Err := FALSE;
   S706_LM_DC_1ST_CLAMP2.M_Ret_Err := FALSE;
   S706_LM_DC_1ST_CLAMP2.LP_Adv := FALSE;
   S706_LM_DC_1ST_CLAMP2.LP_Ret := FALSE;
   S706_LM_DC_1ST_CLAMP2.Visu_Adv := W#16#0;
   S706_LM_DC_1ST_CLAMP2.Visu_Ret := W#16#0;
   S706_LM_DC_1ST_CLAMP2.Error_T1.IN := FALSE;
   S706_LM_DC_1ST_CLAMP2.Error_T1.PT := T#4S;
   S706_LM_DC_1ST_CLAMP2.Error_T1.Q := FALSE;
   S706_LM_DC_1ST_CLAMP2.Error_T1.ET := T#0MS;
   S706_LM_DC_1ST_CLAMP2.Error_T1.STATE := B#16#0;
   S706_LM_DC_1ST_CLAMP2.Error_T1.STIME := T#0MS;
   S706_LM_DC_1ST_CLAMP2.Error_T1.ATIME := T#0MS;
   S706_LM_DC_1ST_CLAMP2.Error_T2.IN := FALSE;
   S706_LM_DC_1ST_CLAMP2.Error_T2.PT := T#4S;
   S706_LM_DC_1ST_CLAMP2.Error_T2.Q := FALSE;
   S706_LM_DC_1ST_CLAMP2.Error_T2.ET := T#0MS;
   S706_LM_DC_1ST_CLAMP2.Error_T2.STATE := B#16#0;
   S706_LM_DC_1ST_CLAMP2.Error_T2.STIME := T#0MS;
   S706_LM_DC_1ST_CLAMP2.Error_T2.ATIME := T#0MS;
   S706_LM_DC_1ST_CLAMP2.CHK_Aux1 := FALSE;
   S706_LM_DC_1ST_CLAMP2.CHK_Aux2 := FALSE;
   S706_LM_DC_1ST_CLAMP2.Error_T1_DN := FALSE;
   S706_LM_DC_1ST_CLAMP2.Error_T2_DN := FALSE;
   S706_LM_DC_1ST_CLAMP2.Adv_Memo := TRUE;
   S706_LM_DC_1ST_CLAMP2.Visu_Adv_Arr[0] := FALSE;
   S706_LM_DC_1ST_CLAMP2.Visu_Adv_Arr[1] := FALSE;
   S706_LM_DC_1ST_CLAMP2.Visu_Adv_Arr[2] := FALSE;
   S706_LM_DC_1ST_CLAMP2.Visu_Adv_Arr[3] := FALSE;
   S706_LM_DC_1ST_CLAMP2.Visu_Adv_Arr[4] := FALSE;
   S706_LM_DC_1ST_CLAMP2.Visu_Adv_Arr[5] := FALSE;
   S706_LM_DC_1ST_CLAMP2.Visu_Adv_Arr[6] := FALSE;
   S706_LM_DC_1ST_CLAMP2.Visu_Adv_Arr[7] := FALSE;
   S706_LM_DC_1ST_CLAMP2.Visu_Adv_Arr[8] := FALSE;
   S706_LM_DC_1ST_CLAMP2.Visu_Adv_Arr[9] := FALSE;
   S706_LM_DC_1ST_CLAMP2.Visu_Adv_Arr[10] := FALSE;
   S706_LM_DC_1ST_CLAMP2.Visu_Adv_Arr[11] := FALSE;
   S706_LM_DC_1ST_CLAMP2.Visu_Adv_Arr[12] := FALSE;
   S706_LM_DC_1ST_CLAMP2.Visu_Adv_Arr[13] := FALSE;
   S706_LM_DC_1ST_CLAMP2.Visu_Adv_Arr[14] := FALSE;
   S706_LM_DC_1ST_CLAMP2.Visu_Adv_Arr[15] := FALSE;
   S706_LM_DC_1ST_CLAMP2.Visu_Ret_Arr[0] := FALSE;
   S706_LM_DC_1ST_CLAMP2.Visu_Ret_Arr[1] := FALSE;
   S706_LM_DC_1ST_CLAMP2.Visu_Ret_Arr[2] := FALSE;
   S706_LM_DC_1ST_CLAMP2.Visu_Ret_Arr[3] := FALSE;
   S706_LM_DC_1ST_CLAMP2.Visu_Ret_Arr[4] := FALSE;
   S706_LM_DC_1ST_CLAMP2.Visu_Ret_Arr[5] := FALSE;
   S706_LM_DC_1ST_CLAMP2.Visu_Ret_Arr[6] := FALSE;
   S706_LM_DC_1ST_CLAMP2.Visu_Ret_Arr[7] := FALSE;
   S706_LM_DC_1ST_CLAMP2.Visu_Ret_Arr[8] := FALSE;
   S706_LM_DC_1ST_CLAMP2.Visu_Ret_Arr[9] := FALSE;
   S706_LM_DC_1ST_CLAMP2.Visu_Ret_Arr[10] := FALSE;
   S706_LM_DC_1ST_CLAMP2.Visu_Ret_Arr[11] := FALSE;
   S706_LM_DC_1ST_CLAMP2.Visu_Ret_Arr[12] := FALSE;
   S706_LM_DC_1ST_CLAMP2.Visu_Ret_Arr[13] := FALSE;
   S706_LM_DC_1ST_CLAMP2.Visu_Ret_Arr[14] := FALSE;
   S706_LM_DC_1ST_CLAMP2.Visu_Ret_Arr[15] := FALSE;
   S706_LM_DC_1ST_CLAMP2.BLK_Move_Ret := 0;
   S706_LM_DC_1ST_CLAMP2.Enable := FALSE;
   S706_LM_DC_1ST_CLAMP2.Adv_End := FALSE;
   S706_LM_DC_1ST_CLAMP2.Ret_End := FALSE;
   S706_LM_DC_1ST_CLAMP3.Enable_Aux := FALSE;
   S706_LM_DC_1ST_CLAMP3.Adv_Amount := 1;
   S706_LM_DC_1ST_CLAMP3.Ret_Amount := 1;
   S706_LM_DC_1ST_CLAMP3.LS_Adv1 := FALSE;
   S706_LM_DC_1ST_CLAMP3.LS_Ret1 := FALSE;
   S706_LM_DC_1ST_CLAMP3.LS_Adv2 := FALSE;
   S706_LM_DC_1ST_CLAMP3.LS_Ret2 := FALSE;
   S706_LM_DC_1ST_CLAMP3.LS_Adv3 := FALSE;
   S706_LM_DC_1ST_CLAMP3.LS_Ret3 := FALSE;
   S706_LM_DC_1ST_CLAMP3.LS_Adv4 := FALSE;
   S706_LM_DC_1ST_CLAMP3.LS_Ret4 := FALSE;
   S706_LM_DC_1ST_CLAMP3.SOL_Adv := FALSE;
   S706_LM_DC_1ST_CLAMP3.SOL_Ret := FALSE;
   S706_LM_DC_1ST_CLAMP3.M_Ready := TRUE;
   S706_LM_DC_1ST_CLAMP3.T_CHK1 := T#4S;
   S706_LM_DC_1ST_CLAMP3.T_CHK2 := T#4S;
   S706_LM_DC_1ST_CLAMP3.PB_Lamp_CHK := FALSE;
   S706_LM_DC_1ST_CLAMP3.PB_Error_Rst := FALSE;
   S706_LM_DC_1ST_CLAMP3.M_FLICK := FALSE;
   S706_LM_DC_1ST_CLAMP3.M_Adv_Err := FALSE;
   S706_LM_DC_1ST_CLAMP3.M_Ret_Err := FALSE;
   S706_LM_DC_1ST_CLAMP3.LP_Adv := FALSE;
   S706_LM_DC_1ST_CLAMP3.LP_Ret := FALSE;
   S706_LM_DC_1ST_CLAMP3.Visu_Adv := W#16#0;
   S706_LM_DC_1ST_CLAMP3.Visu_Ret := W#16#0;
   S706_LM_DC_1ST_CLAMP3.Error_T1.IN := FALSE;
   S706_LM_DC_1ST_CLAMP3.Error_T1.PT := T#4S;
   S706_LM_DC_1ST_CLAMP3.Error_T1.Q := FALSE;
   S706_LM_DC_1ST_CLAMP3.Error_T1.ET := T#0MS;
   S706_LM_DC_1ST_CLAMP3.Error_T1.STATE := B#16#0;
   S706_LM_DC_1ST_CLAMP3.Error_T1.STIME := T#22D22H57M1S422MS;
   S706_LM_DC_1ST_CLAMP3.Error_T1.ATIME := T#22D22H57M1S920MS;
   S706_LM_DC_1ST_CLAMP3.Error_T2.IN := FALSE;
   S706_LM_DC_1ST_CLAMP3.Error_T2.PT := T#4S;
   S706_LM_DC_1ST_CLAMP3.Error_T2.Q := FALSE;
   S706_LM_DC_1ST_CLAMP3.Error_T2.ET := T#0MS;
   S706_LM_DC_1ST_CLAMP3.Error_T2.STATE := B#16#0;
   S706_LM_DC_1ST_CLAMP3.Error_T2.STIME := T#0MS;
   S706_LM_DC_1ST_CLAMP3.Error_T2.ATIME := T#0MS;
   S706_LM_DC_1ST_CLAMP3.CHK_Aux1 := FALSE;
   S706_LM_DC_1ST_CLAMP3.CHK_Aux2 := FALSE;
   S706_LM_DC_1ST_CLAMP3.Error_T1_DN := FALSE;
   S706_LM_DC_1ST_CLAMP3.Error_T2_DN := FALSE;
   S706_LM_DC_1ST_CLAMP3.Adv_Memo := FALSE;
   S706_LM_DC_1ST_CLAMP3.Visu_Adv_Arr[0] := FALSE;
   S706_LM_DC_1ST_CLAMP3.Visu_Adv_Arr[1] := FALSE;
   S706_LM_DC_1ST_CLAMP3.Visu_Adv_Arr[2] := FALSE;
   S706_LM_DC_1ST_CLAMP3.Visu_Adv_Arr[3] := FALSE;
   S706_LM_DC_1ST_CLAMP3.Visu_Adv_Arr[4] := FALSE;
   S706_LM_DC_1ST_CLAMP3.Visu_Adv_Arr[5] := FALSE;
   S706_LM_DC_1ST_CLAMP3.Visu_Adv_Arr[6] := FALSE;
   S706_LM_DC_1ST_CLAMP3.Visu_Adv_Arr[7] := FALSE;
   S706_LM_DC_1ST_CLAMP3.Visu_Adv_Arr[8] := FALSE;
   S706_LM_DC_1ST_CLAMP3.Visu_Adv_Arr[9] := FALSE;
   S706_LM_DC_1ST_CLAMP3.Visu_Adv_Arr[10] := FALSE;
   S706_LM_DC_1ST_CLAMP3.Visu_Adv_Arr[11] := FALSE;
   S706_LM_DC_1ST_CLAMP3.Visu_Adv_Arr[12] := FALSE;
   S706_LM_DC_1ST_CLAMP3.Visu_Adv_Arr[13] := FALSE;
   S706_LM_DC_1ST_CLAMP3.Visu_Adv_Arr[14] := FALSE;
   S706_LM_DC_1ST_CLAMP3.Visu_Adv_Arr[15] := FALSE;
   S706_LM_DC_1ST_CLAMP3.Visu_Ret_Arr[0] := FALSE;
   S706_LM_DC_1ST_CLAMP3.Visu_Ret_Arr[1] := FALSE;
   S706_LM_DC_1ST_CLAMP3.Visu_Ret_Arr[2] := FALSE;
   S706_LM_DC_1ST_CLAMP3.Visu_Ret_Arr[3] := FALSE;
   S706_LM_DC_1ST_CLAMP3.Visu_Ret_Arr[4] := FALSE;
   S706_LM_DC_1ST_CLAMP3.Visu_Ret_Arr[5] := FALSE;
   S706_LM_DC_1ST_CLAMP3.Visu_Ret_Arr[6] := FALSE;
   S706_LM_DC_1ST_CLAMP3.Visu_Ret_Arr[7] := FALSE;
   S706_LM_DC_1ST_CLAMP3.Visu_Ret_Arr[8] := FALSE;
   S706_LM_DC_1ST_CLAMP3.Visu_Ret_Arr[9] := FALSE;
   S706_LM_DC_1ST_CLAMP3.Visu_Ret_Arr[10] := FALSE;
   S706_LM_DC_1ST_CLAMP3.Visu_Ret_Arr[11] := FALSE;
   S706_LM_DC_1ST_CLAMP3.Visu_Ret_Arr[12] := FALSE;
   S706_LM_DC_1ST_CLAMP3.Visu_Ret_Arr[13] := FALSE;
   S706_LM_DC_1ST_CLAMP3.Visu_Ret_Arr[14] := FALSE;
   S706_LM_DC_1ST_CLAMP3.Visu_Ret_Arr[15] := FALSE;
   S706_LM_DC_1ST_CLAMP3.BLK_Move_Ret := 0;
   S706_LM_DC_1ST_CLAMP3.Enable := FALSE;
   S706_LM_DC_1ST_CLAMP3.Adv_End := FALSE;
   S706_LM_DC_1ST_CLAMP3.Ret_End := FALSE;
   S706_LM_DC_1ST_CLAMP4.Enable_Aux := FALSE;
   S706_LM_DC_1ST_CLAMP4.Adv_Amount := 1;
   S706_LM_DC_1ST_CLAMP4.Ret_Amount := 1;
   S706_LM_DC_1ST_CLAMP4.LS_Adv1 := FALSE;
   S706_LM_DC_1ST_CLAMP4.LS_Ret1 := FALSE;
   S706_LM_DC_1ST_CLAMP4.LS_Adv2 := FALSE;
   S706_LM_DC_1ST_CLAMP4.LS_Ret2 := FALSE;
   S706_LM_DC_1ST_CLAMP4.LS_Adv3 := FALSE;
   S706_LM_DC_1ST_CLAMP4.LS_Ret3 := FALSE;
   S706_LM_DC_1ST_CLAMP4.LS_Adv4 := FALSE;
   S706_LM_DC_1ST_CLAMP4.LS_Ret4 := FALSE;
   S706_LM_DC_1ST_CLAMP4.SOL_Adv := FALSE;
   S706_LM_DC_1ST_CLAMP4.SOL_Ret := FALSE;
   S706_LM_DC_1ST_CLAMP4.M_Ready := TRUE;
   S706_LM_DC_1ST_CLAMP4.T_CHK1 := T#4S;
   S706_LM_DC_1ST_CLAMP4.T_CHK2 := T#4S;
   S706_LM_DC_1ST_CLAMP4.PB_Lamp_CHK := FALSE;
   S706_LM_DC_1ST_CLAMP4.PB_Error_Rst := FALSE;
   S706_LM_DC_1ST_CLAMP4.M_FLICK := FALSE;
   S706_LM_DC_1ST_CLAMP4.M_Adv_Err := FALSE;
   S706_LM_DC_1ST_CLAMP4.M_Ret_Err := FALSE;
   S706_LM_DC_1ST_CLAMP4.LP_Adv := FALSE;
   S706_LM_DC_1ST_CLAMP4.LP_Ret := FALSE;
   S706_LM_DC_1ST_CLAMP4.Visu_Adv := W#16#0;
   S706_LM_DC_1ST_CLAMP4.Visu_Ret := W#16#0;
   S706_LM_DC_1ST_CLAMP4.Error_T1.IN := FALSE;
   S706_LM_DC_1ST_CLAMP4.Error_T1.PT := T#4S;
   S706_LM_DC_1ST_CLAMP4.Error_T1.Q := FALSE;
   S706_LM_DC_1ST_CLAMP4.Error_T1.ET := T#0MS;
   S706_LM_DC_1ST_CLAMP4.Error_T1.STATE := B#16#0;
   S706_LM_DC_1ST_CLAMP4.Error_T1.STIME := T#22D22H57M12S190MS;
   S706_LM_DC_1ST_CLAMP4.Error_T1.ATIME := T#22D22H57M12S872MS;
   S706_LM_DC_1ST_CLAMP4.Error_T2.IN := FALSE;
   S706_LM_DC_1ST_CLAMP4.Error_T2.PT := T#4S;
   S706_LM_DC_1ST_CLAMP4.Error_T2.Q := FALSE;
   S706_LM_DC_1ST_CLAMP4.Error_T2.ET := T#0MS;
   S706_LM_DC_1ST_CLAMP4.Error_T2.STATE := B#16#0;
   S706_LM_DC_1ST_CLAMP4.Error_T2.STIME := T#0MS;
   S706_LM_DC_1ST_CLAMP4.Error_T2.ATIME := T#0MS;
   S706_LM_DC_1ST_CLAMP4.CHK_Aux1 := FALSE;
   S706_LM_DC_1ST_CLAMP4.CHK_Aux2 := FALSE;
   S706_LM_DC_1ST_CLAMP4.Error_T1_DN := FALSE;
   S706_LM_DC_1ST_CLAMP4.Error_T2_DN := FALSE;
   S706_LM_DC_1ST_CLAMP4.Adv_Memo := FALSE;
   S706_LM_DC_1ST_CLAMP4.Visu_Adv_Arr[0] := FALSE;
   S706_LM_DC_1ST_CLAMP4.Visu_Adv_Arr[1] := FALSE;
   S706_LM_DC_1ST_CLAMP4.Visu_Adv_Arr[2] := FALSE;
   S706_LM_DC_1ST_CLAMP4.Visu_Adv_Arr[3] := FALSE;
   S706_LM_DC_1ST_CLAMP4.Visu_Adv_Arr[4] := FALSE;
   S706_LM_DC_1ST_CLAMP4.Visu_Adv_Arr[5] := FALSE;
   S706_LM_DC_1ST_CLAMP4.Visu_Adv_Arr[6] := FALSE;
   S706_LM_DC_1ST_CLAMP4.Visu_Adv_Arr[7] := FALSE;
   S706_LM_DC_1ST_CLAMP4.Visu_Adv_Arr[8] := FALSE;
   S706_LM_DC_1ST_CLAMP4.Visu_Adv_Arr[9] := FALSE;
   S706_LM_DC_1ST_CLAMP4.Visu_Adv_Arr[10] := FALSE;
   S706_LM_DC_1ST_CLAMP4.Visu_Adv_Arr[11] := FALSE;
   S706_LM_DC_1ST_CLAMP4.Visu_Adv_Arr[12] := FALSE;
   S706_LM_DC_1ST_CLAMP4.Visu_Adv_Arr[13] := FALSE;
   S706_LM_DC_1ST_CLAMP4.Visu_Adv_Arr[14] := FALSE;
   S706_LM_DC_1ST_CLAMP4.Visu_Adv_Arr[15] := FALSE;
   S706_LM_DC_1ST_CLAMP4.Visu_Ret_Arr[0] := FALSE;
   S706_LM_DC_1ST_CLAMP4.Visu_Ret_Arr[1] := FALSE;
   S706_LM_DC_1ST_CLAMP4.Visu_Ret_Arr[2] := FALSE;
   S706_LM_DC_1ST_CLAMP4.Visu_Ret_Arr[3] := FALSE;
   S706_LM_DC_1ST_CLAMP4.Visu_Ret_Arr[4] := FALSE;
   S706_LM_DC_1ST_CLAMP4.Visu_Ret_Arr[5] := FALSE;
   S706_LM_DC_1ST_CLAMP4.Visu_Ret_Arr[6] := FALSE;
   S706_LM_DC_1ST_CLAMP4.Visu_Ret_Arr[7] := FALSE;
   S706_LM_DC_1ST_CLAMP4.Visu_Ret_Arr[8] := FALSE;
   S706_LM_DC_1ST_CLAMP4.Visu_Ret_Arr[9] := FALSE;
   S706_LM_DC_1ST_CLAMP4.Visu_Ret_Arr[10] := FALSE;
   S706_LM_DC_1ST_CLAMP4.Visu_Ret_Arr[11] := FALSE;
   S706_LM_DC_1ST_CLAMP4.Visu_Ret_Arr[12] := FALSE;
   S706_LM_DC_1ST_CLAMP4.Visu_Ret_Arr[13] := FALSE;
   S706_LM_DC_1ST_CLAMP4.Visu_Ret_Arr[14] := FALSE;
   S706_LM_DC_1ST_CLAMP4.Visu_Ret_Arr[15] := FALSE;
   S706_LM_DC_1ST_CLAMP4.BLK_Move_Ret := 0;
   S706_LM_DC_1ST_CLAMP4.Enable := FALSE;
   S706_LM_DC_1ST_CLAMP4.Adv_End := FALSE;
   S706_LM_DC_1ST_CLAMP4.Ret_End := FALSE;
   S706_LM_DC_2ND_CLAMP1.Enable_Aux := FALSE;
   S706_LM_DC_2ND_CLAMP1.Adv_Amount := 1;
   S706_LM_DC_2ND_CLAMP1.Ret_Amount := 1;
   S706_LM_DC_2ND_CLAMP1.LS_Adv1 := FALSE;
   S706_LM_DC_2ND_CLAMP1.LS_Ret1 := FALSE;
   S706_LM_DC_2ND_CLAMP1.LS_Adv2 := FALSE;
   S706_LM_DC_2ND_CLAMP1.LS_Ret2 := FALSE;
   S706_LM_DC_2ND_CLAMP1.LS_Adv3 := FALSE;
   S706_LM_DC_2ND_CLAMP1.LS_Ret3 := FALSE;
   S706_LM_DC_2ND_CLAMP1.LS_Adv4 := FALSE;
   S706_LM_DC_2ND_CLAMP1.LS_Ret4 := FALSE;
   S706_LM_DC_2ND_CLAMP1.SOL_Adv := FALSE;
   S706_LM_DC_2ND_CLAMP1.SOL_Ret := FALSE;
   S706_LM_DC_2ND_CLAMP1.M_Ready := TRUE;
   S706_LM_DC_2ND_CLAMP1.T_CHK1 := T#4S;
   S706_LM_DC_2ND_CLAMP1.T_CHK2 := T#4S;
   S706_LM_DC_2ND_CLAMP1.PB_Lamp_CHK := FALSE;
   S706_LM_DC_2ND_CLAMP1.PB_Error_Rst := FALSE;
   S706_LM_DC_2ND_CLAMP1.M_FLICK := FALSE;
   S706_LM_DC_2ND_CLAMP1.M_Adv_Err := FALSE;
   S706_LM_DC_2ND_CLAMP1.M_Ret_Err := FALSE;
   S706_LM_DC_2ND_CLAMP1.LP_Adv := FALSE;
   S706_LM_DC_2ND_CLAMP1.LP_Ret := FALSE;
   S706_LM_DC_2ND_CLAMP1.Visu_Adv := W#16#0;
   S706_LM_DC_2ND_CLAMP1.Visu_Ret := W#16#0;
   S706_LM_DC_2ND_CLAMP1.Error_T1.IN := FALSE;
   S706_LM_DC_2ND_CLAMP1.Error_T1.PT := T#4S;
   S706_LM_DC_2ND_CLAMP1.Error_T1.Q := FALSE;
   S706_LM_DC_2ND_CLAMP1.Error_T1.ET := T#0MS;
   S706_LM_DC_2ND_CLAMP1.Error_T1.STATE := B#16#0;
   S706_LM_DC_2ND_CLAMP1.Error_T1.STIME := T#13H10M34S595MS;
   S706_LM_DC_2ND_CLAMP1.Error_T1.ATIME := T#13H10M35S940MS;
   S706_LM_DC_2ND_CLAMP1.Error_T2.IN := FALSE;
   S706_LM_DC_2ND_CLAMP1.Error_T2.PT := T#4S;
   S706_LM_DC_2ND_CLAMP1.Error_T2.Q := FALSE;
   S706_LM_DC_2ND_CLAMP1.Error_T2.ET := T#0MS;
   S706_LM_DC_2ND_CLAMP1.Error_T2.STATE := B#16#0;
   S706_LM_DC_2ND_CLAMP1.Error_T2.STIME := T#0MS;
   S706_LM_DC_2ND_CLAMP1.Error_T2.ATIME := T#0MS;
   S706_LM_DC_2ND_CLAMP1.CHK_Aux1 := FALSE;
   S706_LM_DC_2ND_CLAMP1.CHK_Aux2 := FALSE;
   S706_LM_DC_2ND_CLAMP1.Error_T1_DN := FALSE;
   S706_LM_DC_2ND_CLAMP1.Error_T2_DN := FALSE;
   S706_LM_DC_2ND_CLAMP1.Adv_Memo := TRUE;
   S706_LM_DC_2ND_CLAMP1.Visu_Adv_Arr[0] := FALSE;
   S706_LM_DC_2ND_CLAMP1.Visu_Adv_Arr[1] := FALSE;
   S706_LM_DC_2ND_CLAMP1.Visu_Adv_Arr[2] := FALSE;
   S706_LM_DC_2ND_CLAMP1.Visu_Adv_Arr[3] := FALSE;
   S706_LM_DC_2ND_CLAMP1.Visu_Adv_Arr[4] := FALSE;
   S706_LM_DC_2ND_CLAMP1.Visu_Adv_Arr[5] := FALSE;
   S706_LM_DC_2ND_CLAMP1.Visu_Adv_Arr[6] := FALSE;
   S706_LM_DC_2ND_CLAMP1.Visu_Adv_Arr[7] := FALSE;
   S706_LM_DC_2ND_CLAMP1.Visu_Adv_Arr[8] := FALSE;
   S706_LM_DC_2ND_CLAMP1.Visu_Adv_Arr[9] := FALSE;
   S706_LM_DC_2ND_CLAMP1.Visu_Adv_Arr[10] := FALSE;
   S706_LM_DC_2ND_CLAMP1.Visu_Adv_Arr[11] := FALSE;
   S706_LM_DC_2ND_CLAMP1.Visu_Adv_Arr[12] := FALSE;
   S706_LM_DC_2ND_CLAMP1.Visu_Adv_Arr[13] := FALSE;
   S706_LM_DC_2ND_CLAMP1.Visu_Adv_Arr[14] := FALSE;
   S706_LM_DC_2ND_CLAMP1.Visu_Adv_Arr[15] := FALSE;
   S706_LM_DC_2ND_CLAMP1.Visu_Ret_Arr[0] := FALSE;
   S706_LM_DC_2ND_CLAMP1.Visu_Ret_Arr[1] := FALSE;
   S706_LM_DC_2ND_CLAMP1.Visu_Ret_Arr[2] := FALSE;
   S706_LM_DC_2ND_CLAMP1.Visu_Ret_Arr[3] := FALSE;
   S706_LM_DC_2ND_CLAMP1.Visu_Ret_Arr[4] := FALSE;
   S706_LM_DC_2ND_CLAMP1.Visu_Ret_Arr[5] := FALSE;
   S706_LM_DC_2ND_CLAMP1.Visu_Ret_Arr[6] := FALSE;
   S706_LM_DC_2ND_CLAMP1.Visu_Ret_Arr[7] := FALSE;
   S706_LM_DC_2ND_CLAMP1.Visu_Ret_Arr[8] := FALSE;
   S706_LM_DC_2ND_CLAMP1.Visu_Ret_Arr[9] := FALSE;
   S706_LM_DC_2ND_CLAMP1.Visu_Ret_Arr[10] := FALSE;
   S706_LM_DC_2ND_CLAMP1.Visu_Ret_Arr[11] := FALSE;
   S706_LM_DC_2ND_CLAMP1.Visu_Ret_Arr[12] := FALSE;
   S706_LM_DC_2ND_CLAMP1.Visu_Ret_Arr[13] := FALSE;
   S706_LM_DC_2ND_CLAMP1.Visu_Ret_Arr[14] := FALSE;
   S706_LM_DC_2ND_CLAMP1.Visu_Ret_Arr[15] := FALSE;
   S706_LM_DC_2ND_CLAMP1.BLK_Move_Ret := 0;
   S706_LM_DC_2ND_CLAMP1.Enable := FALSE;
   S706_LM_DC_2ND_CLAMP1.Adv_End := FALSE;
   S706_LM_DC_2ND_CLAMP1.Ret_End := FALSE;
   S706_LM_DC_2ND_CLAMP2.Enable_Aux := FALSE;
   S706_LM_DC_2ND_CLAMP2.Adv_Amount := 1;
   S706_LM_DC_2ND_CLAMP2.Ret_Amount := 1;
   S706_LM_DC_2ND_CLAMP2.LS_Adv1 := FALSE;
   S706_LM_DC_2ND_CLAMP2.LS_Ret1 := FALSE;
   S706_LM_DC_2ND_CLAMP2.LS_Adv2 := FALSE;
   S706_LM_DC_2ND_CLAMP2.LS_Ret2 := FALSE;
   S706_LM_DC_2ND_CLAMP2.LS_Adv3 := FALSE;
   S706_LM_DC_2ND_CLAMP2.LS_Ret3 := FALSE;
   S706_LM_DC_2ND_CLAMP2.LS_Adv4 := FALSE;
   S706_LM_DC_2ND_CLAMP2.LS_Ret4 := FALSE;
   S706_LM_DC_2ND_CLAMP2.SOL_Adv := FALSE;
   S706_LM_DC_2ND_CLAMP2.SOL_Ret := FALSE;
   S706_LM_DC_2ND_CLAMP2.M_Ready := TRUE;
   S706_LM_DC_2ND_CLAMP2.T_CHK1 := T#4S;
   S706_LM_DC_2ND_CLAMP2.T_CHK2 := T#4S;
   S706_LM_DC_2ND_CLAMP2.PB_Lamp_CHK := FALSE;
   S706_LM_DC_2ND_CLAMP2.PB_Error_Rst := FALSE;
   S706_LM_DC_2ND_CLAMP2.M_FLICK := FALSE;
   S706_LM_DC_2ND_CLAMP2.M_Adv_Err := FALSE;
   S706_LM_DC_2ND_CLAMP2.M_Ret_Err := FALSE;
   S706_LM_DC_2ND_CLAMP2.LP_Adv := FALSE;
   S706_LM_DC_2ND_CLAMP2.LP_Ret := FALSE;
   S706_LM_DC_2ND_CLAMP2.Visu_Adv := W#16#0;
   S706_LM_DC_2ND_CLAMP2.Visu_Ret := W#16#0;
   S706_LM_DC_2ND_CLAMP2.Error_T1.IN := FALSE;
   S706_LM_DC_2ND_CLAMP2.Error_T1.PT := T#4S;
   S706_LM_DC_2ND_CLAMP2.Error_T1.Q := FALSE;
   S706_LM_DC_2ND_CLAMP2.Error_T1.ET := T#0MS;
   S706_LM_DC_2ND_CLAMP2.Error_T1.STATE := B#16#0;
   S706_LM_DC_2ND_CLAMP2.Error_T1.STIME := T#12D19H25M56S789MS;
   S706_LM_DC_2ND_CLAMP2.Error_T1.ATIME := T#12D19H25M56S924MS;
   S706_LM_DC_2ND_CLAMP2.Error_T2.IN := FALSE;
   S706_LM_DC_2ND_CLAMP2.Error_T2.PT := T#4S;
   S706_LM_DC_2ND_CLAMP2.Error_T2.Q := FALSE;
   S706_LM_DC_2ND_CLAMP2.Error_T2.ET := T#0MS;
   S706_LM_DC_2ND_CLAMP2.Error_T2.STATE := B#16#0;
   S706_LM_DC_2ND_CLAMP2.Error_T2.STIME := T#0MS;
   S706_LM_DC_2ND_CLAMP2.Error_T2.ATIME := T#0MS;
   S706_LM_DC_2ND_CLAMP2.CHK_Aux1 := FALSE;
   S706_LM_DC_2ND_CLAMP2.CHK_Aux2 := FALSE;
   S706_LM_DC_2ND_CLAMP2.Error_T1_DN := FALSE;
   S706_LM_DC_2ND_CLAMP2.Error_T2_DN := FALSE;
   S706_LM_DC_2ND_CLAMP2.Adv_Memo := TRUE;
   S706_LM_DC_2ND_CLAMP2.Visu_Adv_Arr[0] := FALSE;
   S706_LM_DC_2ND_CLAMP2.Visu_Adv_Arr[1] := FALSE;
   S706_LM_DC_2ND_CLAMP2.Visu_Adv_Arr[2] := FALSE;
   S706_LM_DC_2ND_CLAMP2.Visu_Adv_Arr[3] := FALSE;
   S706_LM_DC_2ND_CLAMP2.Visu_Adv_Arr[4] := FALSE;
   S706_LM_DC_2ND_CLAMP2.Visu_Adv_Arr[5] := FALSE;
   S706_LM_DC_2ND_CLAMP2.Visu_Adv_Arr[6] := FALSE;
   S706_LM_DC_2ND_CLAMP2.Visu_Adv_Arr[7] := FALSE;
   S706_LM_DC_2ND_CLAMP2.Visu_Adv_Arr[8] := FALSE;
   S706_LM_DC_2ND_CLAMP2.Visu_Adv_Arr[9] := FALSE;
   S706_LM_DC_2ND_CLAMP2.Visu_Adv_Arr[10] := FALSE;
   S706_LM_DC_2ND_CLAMP2.Visu_Adv_Arr[11] := FALSE;
   S706_LM_DC_2ND_CLAMP2.Visu_Adv_Arr[12] := FALSE;
   S706_LM_DC_2ND_CLAMP2.Visu_Adv_Arr[13] := FALSE;
   S706_LM_DC_2ND_CLAMP2.Visu_Adv_Arr[14] := FALSE;
   S706_LM_DC_2ND_CLAMP2.Visu_Adv_Arr[15] := FALSE;
   S706_LM_DC_2ND_CLAMP2.Visu_Ret_Arr[0] := FALSE;
   S706_LM_DC_2ND_CLAMP2.Visu_Ret_Arr[1] := FALSE;
   S706_LM_DC_2ND_CLAMP2.Visu_Ret_Arr[2] := FALSE;
   S706_LM_DC_2ND_CLAMP2.Visu_Ret_Arr[3] := FALSE;
   S706_LM_DC_2ND_CLAMP2.Visu_Ret_Arr[4] := FALSE;
   S706_LM_DC_2ND_CLAMP2.Visu_Ret_Arr[5] := FALSE;
   S706_LM_DC_2ND_CLAMP2.Visu_Ret_Arr[6] := FALSE;
   S706_LM_DC_2ND_CLAMP2.Visu_Ret_Arr[7] := FALSE;
   S706_LM_DC_2ND_CLAMP2.Visu_Ret_Arr[8] := FALSE;
   S706_LM_DC_2ND_CLAMP2.Visu_Ret_Arr[9] := FALSE;
   S706_LM_DC_2ND_CLAMP2.Visu_Ret_Arr[10] := FALSE;
   S706_LM_DC_2ND_CLAMP2.Visu_Ret_Arr[11] := FALSE;
   S706_LM_DC_2ND_CLAMP2.Visu_Ret_Arr[12] := FALSE;
   S706_LM_DC_2ND_CLAMP2.Visu_Ret_Arr[13] := FALSE;
   S706_LM_DC_2ND_CLAMP2.Visu_Ret_Arr[14] := FALSE;
   S706_LM_DC_2ND_CLAMP2.Visu_Ret_Arr[15] := FALSE;
   S706_LM_DC_2ND_CLAMP2.BLK_Move_Ret := 0;
   S706_LM_DC_2ND_CLAMP2.Enable := FALSE;
   S706_LM_DC_2ND_CLAMP2.Adv_End := FALSE;
   S706_LM_DC_2ND_CLAMP2.Ret_End := FALSE;
   S706_LM_DC_2ND_CLAMP3.Enable_Aux := FALSE;
   S706_LM_DC_2ND_CLAMP3.Adv_Amount := 1;
   S706_LM_DC_2ND_CLAMP3.Ret_Amount := 1;
   S706_LM_DC_2ND_CLAMP3.LS_Adv1 := FALSE;
   S706_LM_DC_2ND_CLAMP3.LS_Ret1 := FALSE;
   S706_LM_DC_2ND_CLAMP3.LS_Adv2 := FALSE;
   S706_LM_DC_2ND_CLAMP3.LS_Ret2 := FALSE;
   S706_LM_DC_2ND_CLAMP3.LS_Adv3 := FALSE;
   S706_LM_DC_2ND_CLAMP3.LS_Ret3 := FALSE;
   S706_LM_DC_2ND_CLAMP3.LS_Adv4 := FALSE;
   S706_LM_DC_2ND_CLAMP3.LS_Ret4 := FALSE;
   S706_LM_DC_2ND_CLAMP3.SOL_Adv := FALSE;
   S706_LM_DC_2ND_CLAMP3.SOL_Ret := FALSE;
   S706_LM_DC_2ND_CLAMP3.M_Ready := TRUE;
   S706_LM_DC_2ND_CLAMP3.T_CHK1 := T#4S;
   S706_LM_DC_2ND_CLAMP3.T_CHK2 := T#4S;
   S706_LM_DC_2ND_CLAMP3.PB_Lamp_CHK := FALSE;
   S706_LM_DC_2ND_CLAMP3.PB_Error_Rst := FALSE;
   S706_LM_DC_2ND_CLAMP3.M_FLICK := FALSE;
   S706_LM_DC_2ND_CLAMP3.M_Adv_Err := FALSE;
   S706_LM_DC_2ND_CLAMP3.M_Ret_Err := FALSE;
   S706_LM_DC_2ND_CLAMP3.LP_Adv := FALSE;
   S706_LM_DC_2ND_CLAMP3.LP_Ret := FALSE;
   S706_LM_DC_2ND_CLAMP3.Visu_Adv := W#16#0;
   S706_LM_DC_2ND_CLAMP3.Visu_Ret := W#16#0;
   S706_LM_DC_2ND_CLAMP3.Error_T1.IN := FALSE;
   S706_LM_DC_2ND_CLAMP3.Error_T1.PT := T#4S;
   S706_LM_DC_2ND_CLAMP3.Error_T1.Q := FALSE;
   S706_LM_DC_2ND_CLAMP3.Error_T1.ET := T#0MS;
   S706_LM_DC_2ND_CLAMP3.Error_T1.STATE := B#16#0;
   S706_LM_DC_2ND_CLAMP3.Error_T1.STIME := T#0MS;
   S706_LM_DC_2ND_CLAMP3.Error_T1.ATIME := T#0MS;
   S706_LM_DC_2ND_CLAMP3.Error_T2.IN := FALSE;
   S706_LM_DC_2ND_CLAMP3.Error_T2.PT := T#4S;
   S706_LM_DC_2ND_CLAMP3.Error_T2.Q := FALSE;
   S706_LM_DC_2ND_CLAMP3.Error_T2.ET := T#0MS;
   S706_LM_DC_2ND_CLAMP3.Error_T2.STATE := B#16#0;
   S706_LM_DC_2ND_CLAMP3.Error_T2.STIME := T#0MS;
   S706_LM_DC_2ND_CLAMP3.Error_T2.ATIME := T#0MS;
   S706_LM_DC_2ND_CLAMP3.CHK_Aux1 := FALSE;
   S706_LM_DC_2ND_CLAMP3.CHK_Aux2 := FALSE;
   S706_LM_DC_2ND_CLAMP3.Error_T1_DN := FALSE;
   S706_LM_DC_2ND_CLAMP3.Error_T2_DN := FALSE;
   S706_LM_DC_2ND_CLAMP3.Adv_Memo := TRUE;
   S706_LM_DC_2ND_CLAMP3.Visu_Adv_Arr[0] := FALSE;
   S706_LM_DC_2ND_CLAMP3.Visu_Adv_Arr[1] := FALSE;
   S706_LM_DC_2ND_CLAMP3.Visu_Adv_Arr[2] := FALSE;
   S706_LM_DC_2ND_CLAMP3.Visu_Adv_Arr[3] := FALSE;
   S706_LM_DC_2ND_CLAMP3.Visu_Adv_Arr[4] := FALSE;
   S706_LM_DC_2ND_CLAMP3.Visu_Adv_Arr[5] := FALSE;
   S706_LM_DC_2ND_CLAMP3.Visu_Adv_Arr[6] := FALSE;
   S706_LM_DC_2ND_CLAMP3.Visu_Adv_Arr[7] := FALSE;
   S706_LM_DC_2ND_CLAMP3.Visu_Adv_Arr[8] := FALSE;
   S706_LM_DC_2ND_CLAMP3.Visu_Adv_Arr[9] := FALSE;
   S706_LM_DC_2ND_CLAMP3.Visu_Adv_Arr[10] := FALSE;
   S706_LM_DC_2ND_CLAMP3.Visu_Adv_Arr[11] := FALSE;
   S706_LM_DC_2ND_CLAMP3.Visu_Adv_Arr[12] := FALSE;
   S706_LM_DC_2ND_CLAMP3.Visu_Adv_Arr[13] := FALSE;
   S706_LM_DC_2ND_CLAMP3.Visu_Adv_Arr[14] := FALSE;
   S706_LM_DC_2ND_CLAMP3.Visu_Adv_Arr[15] := FALSE;
   S706_LM_DC_2ND_CLAMP3.Visu_Ret_Arr[0] := FALSE;
   S706_LM_DC_2ND_CLAMP3.Visu_Ret_Arr[1] := FALSE;
   S706_LM_DC_2ND_CLAMP3.Visu_Ret_Arr[2] := FALSE;
   S706_LM_DC_2ND_CLAMP3.Visu_Ret_Arr[3] := FALSE;
   S706_LM_DC_2ND_CLAMP3.Visu_Ret_Arr[4] := FALSE;
   S706_LM_DC_2ND_CLAMP3.Visu_Ret_Arr[5] := FALSE;
   S706_LM_DC_2ND_CLAMP3.Visu_Ret_Arr[6] := FALSE;
   S706_LM_DC_2ND_CLAMP3.Visu_Ret_Arr[7] := FALSE;
   S706_LM_DC_2ND_CLAMP3.Visu_Ret_Arr[8] := FALSE;
   S706_LM_DC_2ND_CLAMP3.Visu_Ret_Arr[9] := FALSE;
   S706_LM_DC_2ND_CLAMP3.Visu_Ret_Arr[10] := FALSE;
   S706_LM_DC_2ND_CLAMP3.Visu_Ret_Arr[11] := FALSE;
   S706_LM_DC_2ND_CLAMP3.Visu_Ret_Arr[12] := FALSE;
   S706_LM_DC_2ND_CLAMP3.Visu_Ret_Arr[13] := FALSE;
   S706_LM_DC_2ND_CLAMP3.Visu_Ret_Arr[14] := FALSE;
   S706_LM_DC_2ND_CLAMP3.Visu_Ret_Arr[15] := FALSE;
   S706_LM_DC_2ND_CLAMP3.BLK_Move_Ret := 0;
   S706_LM_DC_2ND_CLAMP3.Enable := FALSE;
   S706_LM_DC_2ND_CLAMP3.Adv_End := FALSE;
   S706_LM_DC_2ND_CLAMP3.Ret_End := FALSE;
   S706_LM_DC_2ND_CLAMP4.Enable_Aux := FALSE;
   S706_LM_DC_2ND_CLAMP4.Adv_Amount := 1;
   S706_LM_DC_2ND_CLAMP4.Ret_Amount := 1;
   S706_LM_DC_2ND_CLAMP4.LS_Adv1 := FALSE;
   S706_LM_DC_2ND_CLAMP4.LS_Ret1 := FALSE;
   S706_LM_DC_2ND_CLAMP4.LS_Adv2 := FALSE;
   S706_LM_DC_2ND_CLAMP4.LS_Ret2 := FALSE;
   S706_LM_DC_2ND_CLAMP4.LS_Adv3 := FALSE;
   S706_LM_DC_2ND_CLAMP4.LS_Ret3 := FALSE;
   S706_LM_DC_2ND_CLAMP4.LS_Adv4 := FALSE;
   S706_LM_DC_2ND_CLAMP4.LS_Ret4 := FALSE;
   S706_LM_DC_2ND_CLAMP4.SOL_Adv := FALSE;
   S706_LM_DC_2ND_CLAMP4.SOL_Ret := FALSE;
   S706_LM_DC_2ND_CLAMP4.M_Ready := TRUE;
   S706_LM_DC_2ND_CLAMP4.T_CHK1 := T#4S;
   S706_LM_DC_2ND_CLAMP4.T_CHK2 := T#4S;
   S706_LM_DC_2ND_CLAMP4.PB_Lamp_CHK := FALSE;
   S706_LM_DC_2ND_CLAMP4.PB_Error_Rst := FALSE;
   S706_LM_DC_2ND_CLAMP4.M_FLICK := FALSE;
   S706_LM_DC_2ND_CLAMP4.M_Adv_Err := FALSE;
   S706_LM_DC_2ND_CLAMP4.M_Ret_Err := FALSE;
   S706_LM_DC_2ND_CLAMP4.LP_Adv := FALSE;
   S706_LM_DC_2ND_CLAMP4.LP_Ret := FALSE;
   S706_LM_DC_2ND_CLAMP4.Visu_Adv := W#16#0;
   S706_LM_DC_2ND_CLAMP4.Visu_Ret := W#16#0;
   S706_LM_DC_2ND_CLAMP4.Error_T1.IN := FALSE;
   S706_LM_DC_2ND_CLAMP4.Error_T1.PT := T#4S;
   S706_LM_DC_2ND_CLAMP4.Error_T1.Q := FALSE;
   S706_LM_DC_2ND_CLAMP4.Error_T1.ET := T#0MS;
   S706_LM_DC_2ND_CLAMP4.Error_T1.STATE := B#16#0;
   S706_LM_DC_2ND_CLAMP4.Error_T1.STIME := T#22D22H57M672MS;
   S706_LM_DC_2ND_CLAMP4.Error_T1.ATIME := T#22D22H57M1S422MS;
   S706_LM_DC_2ND_CLAMP4.Error_T2.IN := FALSE;
   S706_LM_DC_2ND_CLAMP4.Error_T2.PT := T#4S;
   S706_LM_DC_2ND_CLAMP4.Error_T2.Q := FALSE;
   S706_LM_DC_2ND_CLAMP4.Error_T2.ET := T#0MS;
   S706_LM_DC_2ND_CLAMP4.Error_T2.STATE := B#16#0;
   S706_LM_DC_2ND_CLAMP4.Error_T2.STIME := T#0MS;
   S706_LM_DC_2ND_CLAMP4.Error_T2.ATIME := T#0MS;
   S706_LM_DC_2ND_CLAMP4.CHK_Aux1 := FALSE;
   S706_LM_DC_2ND_CLAMP4.CHK_Aux2 := FALSE;
   S706_LM_DC_2ND_CLAMP4.Error_T1_DN := FALSE;
   S706_LM_DC_2ND_CLAMP4.Error_T2_DN := FALSE;
   S706_LM_DC_2ND_CLAMP4.Adv_Memo := FALSE;
   S706_LM_DC_2ND_CLAMP4.Visu_Adv_Arr[0] := FALSE;
   S706_LM_DC_2ND_CLAMP4.Visu_Adv_Arr[1] := FALSE;
   S706_LM_DC_2ND_CLAMP4.Visu_Adv_Arr[2] := FALSE;
   S706_LM_DC_2ND_CLAMP4.Visu_Adv_Arr[3] := FALSE;
   S706_LM_DC_2ND_CLAMP4.Visu_Adv_Arr[4] := FALSE;
   S706_LM_DC_2ND_CLAMP4.Visu_Adv_Arr[5] := FALSE;
   S706_LM_DC_2ND_CLAMP4.Visu_Adv_Arr[6] := FALSE;
   S706_LM_DC_2ND_CLAMP4.Visu_Adv_Arr[7] := FALSE;
   S706_LM_DC_2ND_CLAMP4.Visu_Adv_Arr[8] := FALSE;
   S706_LM_DC_2ND_CLAMP4.Visu_Adv_Arr[9] := FALSE;
   S706_LM_DC_2ND_CLAMP4.Visu_Adv_Arr[10] := FALSE;
   S706_LM_DC_2ND_CLAMP4.Visu_Adv_Arr[11] := FALSE;
   S706_LM_DC_2ND_CLAMP4.Visu_Adv_Arr[12] := FALSE;
   S706_LM_DC_2ND_CLAMP4.Visu_Adv_Arr[13] := FALSE;
   S706_LM_DC_2ND_CLAMP4.Visu_Adv_Arr[14] := FALSE;
   S706_LM_DC_2ND_CLAMP4.Visu_Adv_Arr[15] := FALSE;
   S706_LM_DC_2ND_CLAMP4.Visu_Ret_Arr[0] := FALSE;
   S706_LM_DC_2ND_CLAMP4.Visu_Ret_Arr[1] := FALSE;
   S706_LM_DC_2ND_CLAMP4.Visu_Ret_Arr[2] := FALSE;
   S706_LM_DC_2ND_CLAMP4.Visu_Ret_Arr[3] := FALSE;
   S706_LM_DC_2ND_CLAMP4.Visu_Ret_Arr[4] := FALSE;
   S706_LM_DC_2ND_CLAMP4.Visu_Ret_Arr[5] := FALSE;
   S706_LM_DC_2ND_CLAMP4.Visu_Ret_Arr[6] := FALSE;
   S706_LM_DC_2ND_CLAMP4.Visu_Ret_Arr[7] := FALSE;
   S706_LM_DC_2ND_CLAMP4.Visu_Ret_Arr[8] := FALSE;
   S706_LM_DC_2ND_CLAMP4.Visu_Ret_Arr[9] := FALSE;
   S706_LM_DC_2ND_CLAMP4.Visu_Ret_Arr[10] := FALSE;
   S706_LM_DC_2ND_CLAMP4.Visu_Ret_Arr[11] := FALSE;
   S706_LM_DC_2ND_CLAMP4.Visu_Ret_Arr[12] := FALSE;
   S706_LM_DC_2ND_CLAMP4.Visu_Ret_Arr[13] := FALSE;
   S706_LM_DC_2ND_CLAMP4.Visu_Ret_Arr[14] := FALSE;
   S706_LM_DC_2ND_CLAMP4.Visu_Ret_Arr[15] := FALSE;
   S706_LM_DC_2ND_CLAMP4.BLK_Move_Ret := 0;
   S706_LM_DC_2ND_CLAMP4.Enable := FALSE;
   S706_LM_DC_2ND_CLAMP4.Adv_End := FALSE;
   S706_LM_DC_2ND_CLAMP4.Ret_End := FALSE;
   S706_LM_DC_2ND_CLAMP5.Enable_Aux := FALSE;
   S706_LM_DC_2ND_CLAMP5.Adv_Amount := 1;
   S706_LM_DC_2ND_CLAMP5.Ret_Amount := 1;
   S706_LM_DC_2ND_CLAMP5.LS_Adv1 := FALSE;
   S706_LM_DC_2ND_CLAMP5.LS_Ret1 := FALSE;
   S706_LM_DC_2ND_CLAMP5.LS_Adv2 := FALSE;
   S706_LM_DC_2ND_CLAMP5.LS_Ret2 := FALSE;
   S706_LM_DC_2ND_CLAMP5.LS_Adv3 := FALSE;
   S706_LM_DC_2ND_CLAMP5.LS_Ret3 := FALSE;
   S706_LM_DC_2ND_CLAMP5.LS_Adv4 := FALSE;
   S706_LM_DC_2ND_CLAMP5.LS_Ret4 := FALSE;
   S706_LM_DC_2ND_CLAMP5.SOL_Adv := FALSE;
   S706_LM_DC_2ND_CLAMP5.SOL_Ret := FALSE;
   S706_LM_DC_2ND_CLAMP5.M_Ready := TRUE;
   S706_LM_DC_2ND_CLAMP5.T_CHK1 := T#4S;
   S706_LM_DC_2ND_CLAMP5.T_CHK2 := T#4S;
   S706_LM_DC_2ND_CLAMP5.PB_Lamp_CHK := FALSE;
   S706_LM_DC_2ND_CLAMP5.PB_Error_Rst := FALSE;
   S706_LM_DC_2ND_CLAMP5.M_FLICK := FALSE;
   S706_LM_DC_2ND_CLAMP5.M_Adv_Err := FALSE;
   S706_LM_DC_2ND_CLAMP5.M_Ret_Err := FALSE;
   S706_LM_DC_2ND_CLAMP5.LP_Adv := FALSE;
   S706_LM_DC_2ND_CLAMP5.LP_Ret := FALSE;
   S706_LM_DC_2ND_CLAMP5.Visu_Adv := W#16#0;
   S706_LM_DC_2ND_CLAMP5.Visu_Ret := W#16#0;
   S706_LM_DC_2ND_CLAMP5.Error_T1.IN := FALSE;
   S706_LM_DC_2ND_CLAMP5.Error_T1.PT := T#4S;
   S706_LM_DC_2ND_CLAMP5.Error_T1.Q := FALSE;
   S706_LM_DC_2ND_CLAMP5.Error_T1.ET := T#0MS;
   S706_LM_DC_2ND_CLAMP5.Error_T1.STATE := B#16#0;
   S706_LM_DC_2ND_CLAMP5.Error_T1.STIME := T#22D22H57M10S685MS;
   S706_LM_DC_2ND_CLAMP5.Error_T1.ATIME := T#22D22H57M12S190MS;
   S706_LM_DC_2ND_CLAMP5.Error_T2.IN := FALSE;
   S706_LM_DC_2ND_CLAMP5.Error_T2.PT := T#4S;
   S706_LM_DC_2ND_CLAMP5.Error_T2.Q := FALSE;
   S706_LM_DC_2ND_CLAMP5.Error_T2.ET := T#0MS;
   S706_LM_DC_2ND_CLAMP5.Error_T2.STATE := B#16#0;
   S706_LM_DC_2ND_CLAMP5.Error_T2.STIME := T#0MS;
   S706_LM_DC_2ND_CLAMP5.Error_T2.ATIME := T#0MS;
   S706_LM_DC_2ND_CLAMP5.CHK_Aux1 := FALSE;
   S706_LM_DC_2ND_CLAMP5.CHK_Aux2 := FALSE;
   S706_LM_DC_2ND_CLAMP5.Error_T1_DN := FALSE;
   S706_LM_DC_2ND_CLAMP5.Error_T2_DN := FALSE;
   S706_LM_DC_2ND_CLAMP5.Adv_Memo := FALSE;
   S706_LM_DC_2ND_CLAMP5.Visu_Adv_Arr[0] := FALSE;
   S706_LM_DC_2ND_CLAMP5.Visu_Adv_Arr[1] := FALSE;
   S706_LM_DC_2ND_CLAMP5.Visu_Adv_Arr[2] := FALSE;
   S706_LM_DC_2ND_CLAMP5.Visu_Adv_Arr[3] := FALSE;
   S706_LM_DC_2ND_CLAMP5.Visu_Adv_Arr[4] := FALSE;
   S706_LM_DC_2ND_CLAMP5.Visu_Adv_Arr[5] := FALSE;
   S706_LM_DC_2ND_CLAMP5.Visu_Adv_Arr[6] := FALSE;
   S706_LM_DC_2ND_CLAMP5.Visu_Adv_Arr[7] := FALSE;
   S706_LM_DC_2ND_CLAMP5.Visu_Adv_Arr[8] := FALSE;
   S706_LM_DC_2ND_CLAMP5.Visu_Adv_Arr[9] := FALSE;
   S706_LM_DC_2ND_CLAMP5.Visu_Adv_Arr[10] := FALSE;
   S706_LM_DC_2ND_CLAMP5.Visu_Adv_Arr[11] := FALSE;
   S706_LM_DC_2ND_CLAMP5.Visu_Adv_Arr[12] := FALSE;
   S706_LM_DC_2ND_CLAMP5.Visu_Adv_Arr[13] := FALSE;
   S706_LM_DC_2ND_CLAMP5.Visu_Adv_Arr[14] := FALSE;
   S706_LM_DC_2ND_CLAMP5.Visu_Adv_Arr[15] := FALSE;
   S706_LM_DC_2ND_CLAMP5.Visu_Ret_Arr[0] := FALSE;
   S706_LM_DC_2ND_CLAMP5.Visu_Ret_Arr[1] := FALSE;
   S706_LM_DC_2ND_CLAMP5.Visu_Ret_Arr[2] := FALSE;
   S706_LM_DC_2ND_CLAMP5.Visu_Ret_Arr[3] := FALSE;
   S706_LM_DC_2ND_CLAMP5.Visu_Ret_Arr[4] := FALSE;
   S706_LM_DC_2ND_CLAMP5.Visu_Ret_Arr[5] := FALSE;
   S706_LM_DC_2ND_CLAMP5.Visu_Ret_Arr[6] := FALSE;
   S706_LM_DC_2ND_CLAMP5.Visu_Ret_Arr[7] := FALSE;
   S706_LM_DC_2ND_CLAMP5.Visu_Ret_Arr[8] := FALSE;
   S706_LM_DC_2ND_CLAMP5.Visu_Ret_Arr[9] := FALSE;
   S706_LM_DC_2ND_CLAMP5.Visu_Ret_Arr[10] := FALSE;
   S706_LM_DC_2ND_CLAMP5.Visu_Ret_Arr[11] := FALSE;
   S706_LM_DC_2ND_CLAMP5.Visu_Ret_Arr[12] := FALSE;
   S706_LM_DC_2ND_CLAMP5.Visu_Ret_Arr[13] := FALSE;
   S706_LM_DC_2ND_CLAMP5.Visu_Ret_Arr[14] := FALSE;
   S706_LM_DC_2ND_CLAMP5.Visu_Ret_Arr[15] := FALSE;
   S706_LM_DC_2ND_CLAMP5.BLK_Move_Ret := 0;
   S706_LM_DC_2ND_CLAMP5.Enable := FALSE;
   S706_LM_DC_2ND_CLAMP5.Adv_End := FALSE;
   S706_LM_DC_2ND_CLAMP5.Ret_End := FALSE;
   S706_LM_DC_STK_PIN.Enable_Aux := FALSE;
   S706_LM_DC_STK_PIN.Adv_Amount := 1;
   S706_LM_DC_STK_PIN.Ret_Amount := 1;
   S706_LM_DC_STK_PIN.LS_Adv1 := FALSE;
   S706_LM_DC_STK_PIN.LS_Ret1 := FALSE;
   S706_LM_DC_STK_PIN.LS_Adv2 := FALSE;
   S706_LM_DC_STK_PIN.LS_Ret2 := FALSE;
   S706_LM_DC_STK_PIN.LS_Adv3 := FALSE;
   S706_LM_DC_STK_PIN.LS_Ret3 := FALSE;
   S706_LM_DC_STK_PIN.LS_Adv4 := FALSE;
   S706_LM_DC_STK_PIN.LS_Ret4 := FALSE;
   S706_LM_DC_STK_PIN.SOL_Adv := FALSE;
   S706_LM_DC_STK_PIN.SOL_Ret := FALSE;
   S706_LM_DC_STK_PIN.M_Ready := TRUE;
   S706_LM_DC_STK_PIN.T_CHK1 := T#4S;
   S706_LM_DC_STK_PIN.T_CHK2 := T#4S;
   S706_LM_DC_STK_PIN.PB_Lamp_CHK := FALSE;
   S706_LM_DC_STK_PIN.PB_Error_Rst := FALSE;
   S706_LM_DC_STK_PIN.M_FLICK := FALSE;
   S706_LM_DC_STK_PIN.M_Adv_Err := FALSE;
   S706_LM_DC_STK_PIN.M_Ret_Err := FALSE;
   S706_LM_DC_STK_PIN.LP_Adv := FALSE;
   S706_LM_DC_STK_PIN.LP_Ret := FALSE;
   S706_LM_DC_STK_PIN.Visu_Adv := W#16#0;
   S706_LM_DC_STK_PIN.Visu_Ret := W#16#0;
   S706_LM_DC_STK_PIN.Error_T1.IN := FALSE;
   S706_LM_DC_STK_PIN.Error_T1.PT := T#4S;
   S706_LM_DC_STK_PIN.Error_T1.Q := FALSE;
   S706_LM_DC_STK_PIN.Error_T1.ET := T#0MS;
   S706_LM_DC_STK_PIN.Error_T1.STATE := B#16#0;
   S706_LM_DC_STK_PIN.Error_T1.STIME := T#0MS;
   S706_LM_DC_STK_PIN.Error_T1.ATIME := T#0MS;
   S706_LM_DC_STK_PIN.Error_T2.IN := FALSE;
   S706_LM_DC_STK_PIN.Error_T2.PT := T#4S;
   S706_LM_DC_STK_PIN.Error_T2.Q := FALSE;
   S706_LM_DC_STK_PIN.Error_T2.ET := T#0MS;
   S706_LM_DC_STK_PIN.Error_T2.STATE := B#16#0;
   S706_LM_DC_STK_PIN.Error_T2.STIME := T#0MS;
   S706_LM_DC_STK_PIN.Error_T2.ATIME := T#0MS;
   S706_LM_DC_STK_PIN.CHK_Aux1 := FALSE;
   S706_LM_DC_STK_PIN.CHK_Aux2 := FALSE;
   S706_LM_DC_STK_PIN.Error_T1_DN := FALSE;
   S706_LM_DC_STK_PIN.Error_T2_DN := FALSE;
   S706_LM_DC_STK_PIN.Adv_Memo := FALSE;
   S706_LM_DC_STK_PIN.Visu_Adv_Arr[0] := FALSE;
   S706_LM_DC_STK_PIN.Visu_Adv_Arr[1] := FALSE;
   S706_LM_DC_STK_PIN.Visu_Adv_Arr[2] := FALSE;
   S706_LM_DC_STK_PIN.Visu_Adv_Arr[3] := FALSE;
   S706_LM_DC_STK_PIN.Visu_Adv_Arr[4] := FALSE;
   S706_LM_DC_STK_PIN.Visu_Adv_Arr[5] := FALSE;
   S706_LM_DC_STK_PIN.Visu_Adv_Arr[6] := FALSE;
   S706_LM_DC_STK_PIN.Visu_Adv_Arr[7] := FALSE;
   S706_LM_DC_STK_PIN.Visu_Adv_Arr[8] := FALSE;
   S706_LM_DC_STK_PIN.Visu_Adv_Arr[9] := FALSE;
   S706_LM_DC_STK_PIN.Visu_Adv_Arr[10] := FALSE;
   S706_LM_DC_STK_PIN.Visu_Adv_Arr[11] := FALSE;
   S706_LM_DC_STK_PIN.Visu_Adv_Arr[12] := FALSE;
   S706_LM_DC_STK_PIN.Visu_Adv_Arr[13] := FALSE;
   S706_LM_DC_STK_PIN.Visu_Adv_Arr[14] := FALSE;
   S706_LM_DC_STK_PIN.Visu_Adv_Arr[15] := FALSE;
   S706_LM_DC_STK_PIN.Visu_Ret_Arr[0] := FALSE;
   S706_LM_DC_STK_PIN.Visu_Ret_Arr[1] := FALSE;
   S706_LM_DC_STK_PIN.Visu_Ret_Arr[2] := FALSE;
   S706_LM_DC_STK_PIN.Visu_Ret_Arr[3] := FALSE;
   S706_LM_DC_STK_PIN.Visu_Ret_Arr[4] := FALSE;
   S706_LM_DC_STK_PIN.Visu_Ret_Arr[5] := FALSE;
   S706_LM_DC_STK_PIN.Visu_Ret_Arr[6] := FALSE;
   S706_LM_DC_STK_PIN.Visu_Ret_Arr[7] := FALSE;
   S706_LM_DC_STK_PIN.Visu_Ret_Arr[8] := FALSE;
   S706_LM_DC_STK_PIN.Visu_Ret_Arr[9] := FALSE;
   S706_LM_DC_STK_PIN.Visu_Ret_Arr[10] := FALSE;
   S706_LM_DC_STK_PIN.Visu_Ret_Arr[11] := FALSE;
   S706_LM_DC_STK_PIN.Visu_Ret_Arr[12] := FALSE;
   S706_LM_DC_STK_PIN.Visu_Ret_Arr[13] := FALSE;
   S706_LM_DC_STK_PIN.Visu_Ret_Arr[14] := FALSE;
   S706_LM_DC_STK_PIN.Visu_Ret_Arr[15] := FALSE;
   S706_LM_DC_STK_PIN.BLK_Move_Ret := 0;
   S706_LM_DC_STK_PIN.Enable := FALSE;
   S706_LM_DC_STK_PIN.Adv_End := FALSE;
   S706_LM_DC_STK_PIN.Ret_End := FALSE;
   S706_LM_DC_OTR_CLAMP.Enable_Aux := FALSE;
   S706_LM_DC_OTR_CLAMP.Adv_Amount := 1;
   S706_LM_DC_OTR_CLAMP.Ret_Amount := 1;
   S706_LM_DC_OTR_CLAMP.LS_Adv1 := FALSE;
   S706_LM_DC_OTR_CLAMP.LS_Ret1 := FALSE;
   S706_LM_DC_OTR_CLAMP.LS_Adv2 := FALSE;
   S706_LM_DC_OTR_CLAMP.LS_Ret2 := FALSE;
   S706_LM_DC_OTR_CLAMP.LS_Adv3 := FALSE;
   S706_LM_DC_OTR_CLAMP.LS_Ret3 := FALSE;
   S706_LM_DC_OTR_CLAMP.LS_Adv4 := FALSE;
   S706_LM_DC_OTR_CLAMP.LS_Ret4 := FALSE;
   S706_LM_DC_OTR_CLAMP.SOL_Adv := FALSE;
   S706_LM_DC_OTR_CLAMP.SOL_Ret := FALSE;
   S706_LM_DC_OTR_CLAMP.M_Ready := TRUE;
   S706_LM_DC_OTR_CLAMP.T_CHK1 := T#4S;
   S706_LM_DC_OTR_CLAMP.T_CHK2 := T#4S;
   S706_LM_DC_OTR_CLAMP.PB_Lamp_CHK := FALSE;
   S706_LM_DC_OTR_CLAMP.PB_Error_Rst := FALSE;
   S706_LM_DC_OTR_CLAMP.M_FLICK := FALSE;
   S706_LM_DC_OTR_CLAMP.M_Adv_Err := FALSE;
   S706_LM_DC_OTR_CLAMP.M_Ret_Err := FALSE;
   S706_LM_DC_OTR_CLAMP.LP_Adv := FALSE;
   S706_LM_DC_OTR_CLAMP.LP_Ret := FALSE;
   S706_LM_DC_OTR_CLAMP.Visu_Adv := W#16#0;
   S706_LM_DC_OTR_CLAMP.Visu_Ret := W#16#0;
   S706_LM_DC_OTR_CLAMP.Error_T1.IN := FALSE;
   S706_LM_DC_OTR_CLAMP.Error_T1.PT := T#4S;
   S706_LM_DC_OTR_CLAMP.Error_T1.Q := FALSE;
   S706_LM_DC_OTR_CLAMP.Error_T1.ET := T#0MS;
   S706_LM_DC_OTR_CLAMP.Error_T1.STATE := B#16#0;
   S706_LM_DC_OTR_CLAMP.Error_T1.STIME := T#0MS;
   S706_LM_DC_OTR_CLAMP.Error_T1.ATIME := T#0MS;
   S706_LM_DC_OTR_CLAMP.Error_T2.IN := FALSE;
   S706_LM_DC_OTR_CLAMP.Error_T2.PT := T#4S;
   S706_LM_DC_OTR_CLAMP.Error_T2.Q := FALSE;
   S706_LM_DC_OTR_CLAMP.Error_T2.ET := T#0MS;
   S706_LM_DC_OTR_CLAMP.Error_T2.STATE := B#16#0;
   S706_LM_DC_OTR_CLAMP.Error_T2.STIME := T#0MS;
   S706_LM_DC_OTR_CLAMP.Error_T2.ATIME := T#0MS;
   S706_LM_DC_OTR_CLAMP.CHK_Aux1 := FALSE;
   S706_LM_DC_OTR_CLAMP.CHK_Aux2 := FALSE;
   S706_LM_DC_OTR_CLAMP.Error_T1_DN := FALSE;
   S706_LM_DC_OTR_CLAMP.Error_T2_DN := FALSE;
   S706_LM_DC_OTR_CLAMP.Adv_Memo := FALSE;
   S706_LM_DC_OTR_CLAMP.Visu_Adv_Arr[0] := FALSE;
   S706_LM_DC_OTR_CLAMP.Visu_Adv_Arr[1] := FALSE;
   S706_LM_DC_OTR_CLAMP.Visu_Adv_Arr[2] := FALSE;
   S706_LM_DC_OTR_CLAMP.Visu_Adv_Arr[3] := FALSE;
   S706_LM_DC_OTR_CLAMP.Visu_Adv_Arr[4] := FALSE;
   S706_LM_DC_OTR_CLAMP.Visu_Adv_Arr[5] := FALSE;
   S706_LM_DC_OTR_CLAMP.Visu_Adv_Arr[6] := FALSE;
   S706_LM_DC_OTR_CLAMP.Visu_Adv_Arr[7] := FALSE;
   S706_LM_DC_OTR_CLAMP.Visu_Adv_Arr[8] := FALSE;
   S706_LM_DC_OTR_CLAMP.Visu_Adv_Arr[9] := FALSE;
   S706_LM_DC_OTR_CLAMP.Visu_Adv_Arr[10] := FALSE;
   S706_LM_DC_OTR_CLAMP.Visu_Adv_Arr[11] := FALSE;
   S706_LM_DC_OTR_CLAMP.Visu_Adv_Arr[12] := FALSE;
   S706_LM_DC_OTR_CLAMP.Visu_Adv_Arr[13] := FALSE;
   S706_LM_DC_OTR_CLAMP.Visu_Adv_Arr[14] := FALSE;
   S706_LM_DC_OTR_CLAMP.Visu_Adv_Arr[15] := FALSE;
   S706_LM_DC_OTR_CLAMP.Visu_Ret_Arr[0] := FALSE;
   S706_LM_DC_OTR_CLAMP.Visu_Ret_Arr[1] := FALSE;
   S706_LM_DC_OTR_CLAMP.Visu_Ret_Arr[2] := FALSE;
   S706_LM_DC_OTR_CLAMP.Visu_Ret_Arr[3] := FALSE;
   S706_LM_DC_OTR_CLAMP.Visu_Ret_Arr[4] := FALSE;
   S706_LM_DC_OTR_CLAMP.Visu_Ret_Arr[5] := FALSE;
   S706_LM_DC_OTR_CLAMP.Visu_Ret_Arr[6] := FALSE;
   S706_LM_DC_OTR_CLAMP.Visu_Ret_Arr[7] := FALSE;
   S706_LM_DC_OTR_CLAMP.Visu_Ret_Arr[8] := FALSE;
   S706_LM_DC_OTR_CLAMP.Visu_Ret_Arr[9] := FALSE;
   S706_LM_DC_OTR_CLAMP.Visu_Ret_Arr[10] := FALSE;
   S706_LM_DC_OTR_CLAMP.Visu_Ret_Arr[11] := FALSE;
   S706_LM_DC_OTR_CLAMP.Visu_Ret_Arr[12] := FALSE;
   S706_LM_DC_OTR_CLAMP.Visu_Ret_Arr[13] := FALSE;
   S706_LM_DC_OTR_CLAMP.Visu_Ret_Arr[14] := FALSE;
   S706_LM_DC_OTR_CLAMP.Visu_Ret_Arr[15] := FALSE;
   S706_LM_DC_OTR_CLAMP.BLK_Move_Ret := 0;
   S706_LM_DC_OTR_CLAMP.Enable := FALSE;
   S706_LM_DC_OTR_CLAMP.Adv_End := FALSE;
   S706_LM_DC_OTR_CLAMP.Ret_End := FALSE;
   S706_LM_DC_ASSY_CLAMP.Enable_Aux := FALSE;
   S706_LM_DC_ASSY_CLAMP.Adv_Amount := 1;
   S706_LM_DC_ASSY_CLAMP.Ret_Amount := 1;
   S706_LM_DC_ASSY_CLAMP.LS_Adv1 := FALSE;
   S706_LM_DC_ASSY_CLAMP.LS_Ret1 := FALSE;
   S706_LM_DC_ASSY_CLAMP.LS_Adv2 := FALSE;
   S706_LM_DC_ASSY_CLAMP.LS_Ret2 := FALSE;
   S706_LM_DC_ASSY_CLAMP.LS_Adv3 := FALSE;
   S706_LM_DC_ASSY_CLAMP.LS_Ret3 := FALSE;
   S706_LM_DC_ASSY_CLAMP.LS_Adv4 := FALSE;
   S706_LM_DC_ASSY_CLAMP.LS_Ret4 := FALSE;
   S706_LM_DC_ASSY_CLAMP.SOL_Adv := FALSE;
   S706_LM_DC_ASSY_CLAMP.SOL_Ret := FALSE;
   S706_LM_DC_ASSY_CLAMP.M_Ready := TRUE;
   S706_LM_DC_ASSY_CLAMP.T_CHK1 := T#4S;
   S706_LM_DC_ASSY_CLAMP.T_CHK2 := T#4S;
   S706_LM_DC_ASSY_CLAMP.PB_Lamp_CHK := FALSE;
   S706_LM_DC_ASSY_CLAMP.PB_Error_Rst := FALSE;
   S706_LM_DC_ASSY_CLAMP.M_FLICK := FALSE;
   S706_LM_DC_ASSY_CLAMP.M_Adv_Err := FALSE;
   S706_LM_DC_ASSY_CLAMP.M_Ret_Err := FALSE;
   S706_LM_DC_ASSY_CLAMP.LP_Adv := FALSE;
   S706_LM_DC_ASSY_CLAMP.LP_Ret := FALSE;
   S706_LM_DC_ASSY_CLAMP.Visu_Adv := W#16#0;
   S706_LM_DC_ASSY_CLAMP.Visu_Ret := W#16#0;
   S706_LM_DC_ASSY_CLAMP.Error_T1.IN := FALSE;
   S706_LM_DC_ASSY_CLAMP.Error_T1.PT := T#4S;
   S706_LM_DC_ASSY_CLAMP.Error_T1.Q := FALSE;
   S706_LM_DC_ASSY_CLAMP.Error_T1.ET := T#0MS;
   S706_LM_DC_ASSY_CLAMP.Error_T1.STATE := B#16#0;
   S706_LM_DC_ASSY_CLAMP.Error_T1.STIME := T#0MS;
   S706_LM_DC_ASSY_CLAMP.Error_T1.ATIME := T#0MS;
   S706_LM_DC_ASSY_CLAMP.Error_T2.IN := FALSE;
   S706_LM_DC_ASSY_CLAMP.Error_T2.PT := T#4S;
   S706_LM_DC_ASSY_CLAMP.Error_T2.Q := FALSE;
   S706_LM_DC_ASSY_CLAMP.Error_T2.ET := T#0MS;
   S706_LM_DC_ASSY_CLAMP.Error_T2.STATE := B#16#0;
   S706_LM_DC_ASSY_CLAMP.Error_T2.STIME := T#0MS;
   S706_LM_DC_ASSY_CLAMP.Error_T2.ATIME := T#0MS;
   S706_LM_DC_ASSY_CLAMP.CHK_Aux1 := FALSE;
   S706_LM_DC_ASSY_CLAMP.CHK_Aux2 := FALSE;
   S706_LM_DC_ASSY_CLAMP.Error_T1_DN := FALSE;
   S706_LM_DC_ASSY_CLAMP.Error_T2_DN := FALSE;
   S706_LM_DC_ASSY_CLAMP.Adv_Memo := TRUE;
   S706_LM_DC_ASSY_CLAMP.Visu_Adv_Arr[0] := FALSE;
   S706_LM_DC_ASSY_CLAMP.Visu_Adv_Arr[1] := FALSE;
   S706_LM_DC_ASSY_CLAMP.Visu_Adv_Arr[2] := FALSE;
   S706_LM_DC_ASSY_CLAMP.Visu_Adv_Arr[3] := FALSE;
   S706_LM_DC_ASSY_CLAMP.Visu_Adv_Arr[4] := FALSE;
   S706_LM_DC_ASSY_CLAMP.Visu_Adv_Arr[5] := FALSE;
   S706_LM_DC_ASSY_CLAMP.Visu_Adv_Arr[6] := FALSE;
   S706_LM_DC_ASSY_CLAMP.Visu_Adv_Arr[7] := FALSE;
   S706_LM_DC_ASSY_CLAMP.Visu_Adv_Arr[8] := FALSE;
   S706_LM_DC_ASSY_CLAMP.Visu_Adv_Arr[9] := FALSE;
   S706_LM_DC_ASSY_CLAMP.Visu_Adv_Arr[10] := FALSE;
   S706_LM_DC_ASSY_CLAMP.Visu_Adv_Arr[11] := FALSE;
   S706_LM_DC_ASSY_CLAMP.Visu_Adv_Arr[12] := FALSE;
   S706_LM_DC_ASSY_CLAMP.Visu_Adv_Arr[13] := FALSE;
   S706_LM_DC_ASSY_CLAMP.Visu_Adv_Arr[14] := FALSE;
   S706_LM_DC_ASSY_CLAMP.Visu_Adv_Arr[15] := FALSE;
   S706_LM_DC_ASSY_CLAMP.Visu_Ret_Arr[0] := FALSE;
   S706_LM_DC_ASSY_CLAMP.Visu_Ret_Arr[1] := FALSE;
   S706_LM_DC_ASSY_CLAMP.Visu_Ret_Arr[2] := FALSE;
   S706_LM_DC_ASSY_CLAMP.Visu_Ret_Arr[3] := FALSE;
   S706_LM_DC_ASSY_CLAMP.Visu_Ret_Arr[4] := FALSE;
   S706_LM_DC_ASSY_CLAMP.Visu_Ret_Arr[5] := FALSE;
   S706_LM_DC_ASSY_CLAMP.Visu_Ret_Arr[6] := FALSE;
   S706_LM_DC_ASSY_CLAMP.Visu_Ret_Arr[7] := FALSE;
   S706_LM_DC_ASSY_CLAMP.Visu_Ret_Arr[8] := FALSE;
   S706_LM_DC_ASSY_CLAMP.Visu_Ret_Arr[9] := FALSE;
   S706_LM_DC_ASSY_CLAMP.Visu_Ret_Arr[10] := FALSE;
   S706_LM_DC_ASSY_CLAMP.Visu_Ret_Arr[11] := FALSE;
   S706_LM_DC_ASSY_CLAMP.Visu_Ret_Arr[12] := FALSE;
   S706_LM_DC_ASSY_CLAMP.Visu_Ret_Arr[13] := FALSE;
   S706_LM_DC_ASSY_CLAMP.Visu_Ret_Arr[14] := FALSE;
   S706_LM_DC_ASSY_CLAMP.Visu_Ret_Arr[15] := FALSE;
   S706_LM_DC_ASSY_CLAMP.BLK_Move_Ret := 0;
   S706_LM_DC_ASSY_CLAMP.Enable := FALSE;
   S706_LM_DC_ASSY_CLAMP.Adv_End := FALSE;
   S706_LM_DC_ASSY_CLAMP.Ret_End := FALSE;
   S706_LM_DC_FF_PIN.Enable_Aux := FALSE;
   S706_LM_DC_FF_PIN.Adv_Amount := 1;
   S706_LM_DC_FF_PIN.Ret_Amount := 1;
   S706_LM_DC_FF_PIN.LS_Adv1 := FALSE;
   S706_LM_DC_FF_PIN.LS_Ret1 := FALSE;
   S706_LM_DC_FF_PIN.LS_Adv2 := FALSE;
   S706_LM_DC_FF_PIN.LS_Ret2 := FALSE;
   S706_LM_DC_FF_PIN.LS_Adv3 := FALSE;
   S706_LM_DC_FF_PIN.LS_Ret3 := FALSE;
   S706_LM_DC_FF_PIN.LS_Adv4 := FALSE;
   S706_LM_DC_FF_PIN.LS_Ret4 := FALSE;
   S706_LM_DC_FF_PIN.SOL_Adv := FALSE;
   S706_LM_DC_FF_PIN.SOL_Ret := FALSE;
   S706_LM_DC_FF_PIN.M_Ready := TRUE;
   S706_LM_DC_FF_PIN.T_CHK1 := T#4S;
   S706_LM_DC_FF_PIN.T_CHK2 := T#4S;
   S706_LM_DC_FF_PIN.PB_Lamp_CHK := FALSE;
   S706_LM_DC_FF_PIN.PB_Error_Rst := FALSE;
   S706_LM_DC_FF_PIN.M_FLICK := FALSE;
   S706_LM_DC_FF_PIN.M_Adv_Err := FALSE;
   S706_LM_DC_FF_PIN.M_Ret_Err := FALSE;
   S706_LM_DC_FF_PIN.LP_Adv := FALSE;
   S706_LM_DC_FF_PIN.LP_Ret := FALSE;
   S706_LM_DC_FF_PIN.Visu_Adv := W#16#0;
   S706_LM_DC_FF_PIN.Visu_Ret := W#16#0;
   S706_LM_DC_FF_PIN.Error_T1.IN := FALSE;
   S706_LM_DC_FF_PIN.Error_T1.PT := T#4S;
   S706_LM_DC_FF_PIN.Error_T1.Q := FALSE;
   S706_LM_DC_FF_PIN.Error_T1.ET := T#0MS;
   S706_LM_DC_FF_PIN.Error_T1.STATE := B#16#0;
   S706_LM_DC_FF_PIN.Error_T1.STIME := T#0MS;
   S706_LM_DC_FF_PIN.Error_T1.ATIME := T#0MS;
   S706_LM_DC_FF_PIN.Error_T2.IN := FALSE;
   S706_LM_DC_FF_PIN.Error_T2.PT := T#4S;
   S706_LM_DC_FF_PIN.Error_T2.Q := FALSE;
   S706_LM_DC_FF_PIN.Error_T2.ET := T#0MS;
   S706_LM_DC_FF_PIN.Error_T2.STATE := B#16#0;
   S706_LM_DC_FF_PIN.Error_T2.STIME := T#0MS;
   S706_LM_DC_FF_PIN.Error_T2.ATIME := T#0MS;
   S706_LM_DC_FF_PIN.CHK_Aux1 := FALSE;
   S706_LM_DC_FF_PIN.CHK_Aux2 := FALSE;
   S706_LM_DC_FF_PIN.Error_T1_DN := FALSE;
   S706_LM_DC_FF_PIN.Error_T2_DN := FALSE;
   S706_LM_DC_FF_PIN.Adv_Memo := FALSE;
   S706_LM_DC_FF_PIN.Visu_Adv_Arr[0] := FALSE;
   S706_LM_DC_FF_PIN.Visu_Adv_Arr[1] := FALSE;
   S706_LM_DC_FF_PIN.Visu_Adv_Arr[2] := FALSE;
   S706_LM_DC_FF_PIN.Visu_Adv_Arr[3] := FALSE;
   S706_LM_DC_FF_PIN.Visu_Adv_Arr[4] := FALSE;
   S706_LM_DC_FF_PIN.Visu_Adv_Arr[5] := FALSE;
   S706_LM_DC_FF_PIN.Visu_Adv_Arr[6] := FALSE;
   S706_LM_DC_FF_PIN.Visu_Adv_Arr[7] := FALSE;
   S706_LM_DC_FF_PIN.Visu_Adv_Arr[8] := FALSE;
   S706_LM_DC_FF_PIN.Visu_Adv_Arr[9] := FALSE;
   S706_LM_DC_FF_PIN.Visu_Adv_Arr[10] := FALSE;
   S706_LM_DC_FF_PIN.Visu_Adv_Arr[11] := FALSE;
   S706_LM_DC_FF_PIN.Visu_Adv_Arr[12] := FALSE;
   S706_LM_DC_FF_PIN.Visu_Adv_Arr[13] := FALSE;
   S706_LM_DC_FF_PIN.Visu_Adv_Arr[14] := FALSE;
   S706_LM_DC_FF_PIN.Visu_Adv_Arr[15] := FALSE;
   S706_LM_DC_FF_PIN.Visu_Ret_Arr[0] := FALSE;
   S706_LM_DC_FF_PIN.Visu_Ret_Arr[1] := FALSE;
   S706_LM_DC_FF_PIN.Visu_Ret_Arr[2] := FALSE;
   S706_LM_DC_FF_PIN.Visu_Ret_Arr[3] := FALSE;
   S706_LM_DC_FF_PIN.Visu_Ret_Arr[4] := FALSE;
   S706_LM_DC_FF_PIN.Visu_Ret_Arr[5] := FALSE;
   S706_LM_DC_FF_PIN.Visu_Ret_Arr[6] := FALSE;
   S706_LM_DC_FF_PIN.Visu_Ret_Arr[7] := FALSE;
   S706_LM_DC_FF_PIN.Visu_Ret_Arr[8] := FALSE;
   S706_LM_DC_FF_PIN.Visu_Ret_Arr[9] := FALSE;
   S706_LM_DC_FF_PIN.Visu_Ret_Arr[10] := FALSE;
   S706_LM_DC_FF_PIN.Visu_Ret_Arr[11] := FALSE;
   S706_LM_DC_FF_PIN.Visu_Ret_Arr[12] := FALSE;
   S706_LM_DC_FF_PIN.Visu_Ret_Arr[13] := FALSE;
   S706_LM_DC_FF_PIN.Visu_Ret_Arr[14] := FALSE;
   S706_LM_DC_FF_PIN.Visu_Ret_Arr[15] := FALSE;
   S706_LM_DC_FF_PIN.BLK_Move_Ret := 0;
   S706_LM_DC_FF_PIN.Enable := FALSE;
   S706_LM_DC_FF_PIN.Adv_End := FALSE;
   S706_LM_DC_FF_PIN.Ret_End := FALSE;
   S706_LM_DC_FF_CLAMP.Enable_Aux := FALSE;
   S706_LM_DC_FF_CLAMP.Adv_Amount := 1;
   S706_LM_DC_FF_CLAMP.Ret_Amount := 1;
   S706_LM_DC_FF_CLAMP.LS_Adv1 := FALSE;
   S706_LM_DC_FF_CLAMP.LS_Ret1 := FALSE;
   S706_LM_DC_FF_CLAMP.LS_Adv2 := FALSE;
   S706_LM_DC_FF_CLAMP.LS_Ret2 := FALSE;
   S706_LM_DC_FF_CLAMP.LS_Adv3 := FALSE;
   S706_LM_DC_FF_CLAMP.LS_Ret3 := FALSE;
   S706_LM_DC_FF_CLAMP.LS_Adv4 := FALSE;
   S706_LM_DC_FF_CLAMP.LS_Ret4 := FALSE;
   S706_LM_DC_FF_CLAMP.SOL_Adv := FALSE;
   S706_LM_DC_FF_CLAMP.SOL_Ret := FALSE;
   S706_LM_DC_FF_CLAMP.M_Ready := TRUE;
   S706_LM_DC_FF_CLAMP.T_CHK1 := T#4S;
   S706_LM_DC_FF_CLAMP.T_CHK2 := T#4S;
   S706_LM_DC_FF_CLAMP.PB_Lamp_CHK := FALSE;
   S706_LM_DC_FF_CLAMP.PB_Error_Rst := FALSE;
   S706_LM_DC_FF_CLAMP.M_FLICK := FALSE;
   S706_LM_DC_FF_CLAMP.M_Adv_Err := FALSE;
   S706_LM_DC_FF_CLAMP.M_Ret_Err := FALSE;
   S706_LM_DC_FF_CLAMP.LP_Adv := FALSE;
   S706_LM_DC_FF_CLAMP.LP_Ret := FALSE;
   S706_LM_DC_FF_CLAMP.Visu_Adv := W#16#0;
   S706_LM_DC_FF_CLAMP.Visu_Ret := W#16#0;
   S706_LM_DC_FF_CLAMP.Error_T1.IN := FALSE;
   S706_LM_DC_FF_CLAMP.Error_T1.PT := T#4S;
   S706_LM_DC_FF_CLAMP.Error_T1.Q := FALSE;
   S706_LM_DC_FF_CLAMP.Error_T1.ET := T#0MS;
   S706_LM_DC_FF_CLAMP.Error_T1.STATE := B#16#0;
   S706_LM_DC_FF_CLAMP.Error_T1.STIME := T#0MS;
   S706_LM_DC_FF_CLAMP.Error_T1.ATIME := T#0MS;
   S706_LM_DC_FF_CLAMP.Error_T2.IN := FALSE;
   S706_LM_DC_FF_CLAMP.Error_T2.PT := T#4S;
   S706_LM_DC_FF_CLAMP.Error_T2.Q := FALSE;
   S706_LM_DC_FF_CLAMP.Error_T2.ET := T#0MS;
   S706_LM_DC_FF_CLAMP.Error_T2.STATE := B#16#0;
   S706_LM_DC_FF_CLAMP.Error_T2.STIME := T#0MS;
   S706_LM_DC_FF_CLAMP.Error_T2.ATIME := T#0MS;
   S706_LM_DC_FF_CLAMP.CHK_Aux1 := FALSE;
   S706_LM_DC_FF_CLAMP.CHK_Aux2 := FALSE;
   S706_LM_DC_FF_CLAMP.Error_T1_DN := FALSE;
   S706_LM_DC_FF_CLAMP.Error_T2_DN := FALSE;
   S706_LM_DC_FF_CLAMP.Adv_Memo := FALSE;
   S706_LM_DC_FF_CLAMP.Visu_Adv_Arr[0] := FALSE;
   S706_LM_DC_FF_CLAMP.Visu_Adv_Arr[1] := FALSE;
   S706_LM_DC_FF_CLAMP.Visu_Adv_Arr[2] := FALSE;
   S706_LM_DC_FF_CLAMP.Visu_Adv_Arr[3] := FALSE;
   S706_LM_DC_FF_CLAMP.Visu_Adv_Arr[4] := FALSE;
   S706_LM_DC_FF_CLAMP.Visu_Adv_Arr[5] := FALSE;
   S706_LM_DC_FF_CLAMP.Visu_Adv_Arr[6] := FALSE;
   S706_LM_DC_FF_CLAMP.Visu_Adv_Arr[7] := FALSE;
   S706_LM_DC_FF_CLAMP.Visu_Adv_Arr[8] := FALSE;
   S706_LM_DC_FF_CLAMP.Visu_Adv_Arr[9] := FALSE;
   S706_LM_DC_FF_CLAMP.Visu_Adv_Arr[10] := FALSE;
   S706_LM_DC_FF_CLAMP.Visu_Adv_Arr[11] := FALSE;
   S706_LM_DC_FF_CLAMP.Visu_Adv_Arr[12] := FALSE;
   S706_LM_DC_FF_CLAMP.Visu_Adv_Arr[13] := FALSE;
   S706_LM_DC_FF_CLAMP.Visu_Adv_Arr[14] := FALSE;
   S706_LM_DC_FF_CLAMP.Visu_Adv_Arr[15] := FALSE;
   S706_LM_DC_FF_CLAMP.Visu_Ret_Arr[0] := FALSE;
   S706_LM_DC_FF_CLAMP.Visu_Ret_Arr[1] := FALSE;
   S706_LM_DC_FF_CLAMP.Visu_Ret_Arr[2] := FALSE;
   S706_LM_DC_FF_CLAMP.Visu_Ret_Arr[3] := FALSE;
   S706_LM_DC_FF_CLAMP.Visu_Ret_Arr[4] := FALSE;
   S706_LM_DC_FF_CLAMP.Visu_Ret_Arr[5] := FALSE;
   S706_LM_DC_FF_CLAMP.Visu_Ret_Arr[6] := FALSE;
   S706_LM_DC_FF_CLAMP.Visu_Ret_Arr[7] := FALSE;
   S706_LM_DC_FF_CLAMP.Visu_Ret_Arr[8] := FALSE;
   S706_LM_DC_FF_CLAMP.Visu_Ret_Arr[9] := FALSE;
   S706_LM_DC_FF_CLAMP.Visu_Ret_Arr[10] := FALSE;
   S706_LM_DC_FF_CLAMP.Visu_Ret_Arr[11] := FALSE;
   S706_LM_DC_FF_CLAMP.Visu_Ret_Arr[12] := FALSE;
   S706_LM_DC_FF_CLAMP.Visu_Ret_Arr[13] := FALSE;
   S706_LM_DC_FF_CLAMP.Visu_Ret_Arr[14] := FALSE;
   S706_LM_DC_FF_CLAMP.Visu_Ret_Arr[15] := FALSE;
   S706_LM_DC_FF_CLAMP.BLK_Move_Ret := 0;
   S706_LM_DC_FF_CLAMP.Enable := FALSE;
   S706_LM_DC_FF_CLAMP.Adv_End := FALSE;
   S706_LM_DC_FF_CLAMP.Ret_End := FALSE;
   S706_LM_DC_2ND_CLAMP6.Enable_Aux := FALSE;
   S706_LM_DC_2ND_CLAMP6.Adv_Amount := 2;
   S706_LM_DC_2ND_CLAMP6.Ret_Amount := 2;
   S706_LM_DC_2ND_CLAMP6.LS_Adv1 := FALSE;
   S706_LM_DC_2ND_CLAMP6.LS_Ret1 := FALSE;
   S706_LM_DC_2ND_CLAMP6.LS_Adv2 := FALSE;
   S706_LM_DC_2ND_CLAMP6.LS_Ret2 := FALSE;
   S706_LM_DC_2ND_CLAMP6.LS_Adv3 := FALSE;
   S706_LM_DC_2ND_CLAMP6.LS_Ret3 := FALSE;
   S706_LM_DC_2ND_CLAMP6.LS_Adv4 := FALSE;
   S706_LM_DC_2ND_CLAMP6.LS_Ret4 := FALSE;
   S706_LM_DC_2ND_CLAMP6.SOL_Adv := FALSE;
   S706_LM_DC_2ND_CLAMP6.SOL_Ret := FALSE;
   S706_LM_DC_2ND_CLAMP6.M_Ready := TRUE;
   S706_LM_DC_2ND_CLAMP6.T_CHK1 := T#4S;
   S706_LM_DC_2ND_CLAMP6.T_CHK2 := T#4S;
   S706_LM_DC_2ND_CLAMP6.PB_Lamp_CHK := FALSE;
   S706_LM_DC_2ND_CLAMP6.PB_Error_Rst := FALSE;
   S706_LM_DC_2ND_CLAMP6.M_FLICK := FALSE;
   S706_LM_DC_2ND_CLAMP6.M_Adv_Err := FALSE;
   S706_LM_DC_2ND_CLAMP6.M_Ret_Err := FALSE;
   S706_LM_DC_2ND_CLAMP6.LP_Adv := FALSE;
   S706_LM_DC_2ND_CLAMP6.LP_Ret := FALSE;
   S706_LM_DC_2ND_CLAMP6.Visu_Adv := W#16#0;
   S706_LM_DC_2ND_CLAMP6.Visu_Ret := W#16#0;
   S706_LM_DC_2ND_CLAMP6.Error_T1.IN := FALSE;
   S706_LM_DC_2ND_CLAMP6.Error_T1.PT := T#4S;
   S706_LM_DC_2ND_CLAMP6.Error_T1.Q := FALSE;
   S706_LM_DC_2ND_CLAMP6.Error_T1.ET := T#0MS;
   S706_LM_DC_2ND_CLAMP6.Error_T1.STATE := B#16#0;
   S706_LM_DC_2ND_CLAMP6.Error_T1.STIME := T#0MS;
   S706_LM_DC_2ND_CLAMP6.Error_T1.ATIME := T#0MS;
   S706_LM_DC_2ND_CLAMP6.Error_T2.IN := FALSE;
   S706_LM_DC_2ND_CLAMP6.Error_T2.PT := T#4S;
   S706_LM_DC_2ND_CLAMP6.Error_T2.Q := FALSE;
   S706_LM_DC_2ND_CLAMP6.Error_T2.ET := T#0MS;
   S706_LM_DC_2ND_CLAMP6.Error_T2.STATE := B#16#0;
   S706_LM_DC_2ND_CLAMP6.Error_T2.STIME := T#0MS;
   S706_LM_DC_2ND_CLAMP6.Error_T2.ATIME := T#0MS;
   S706_LM_DC_2ND_CLAMP6.CHK_Aux1 := FALSE;
   S706_LM_DC_2ND_CLAMP6.CHK_Aux2 := FALSE;
   S706_LM_DC_2ND_CLAMP6.Error_T1_DN := FALSE;
   S706_LM_DC_2ND_CLAMP6.Error_T2_DN := FALSE;
   S706_LM_DC_2ND_CLAMP6.Adv_Memo := TRUE;
   S706_LM_DC_2ND_CLAMP6.Visu_Adv_Arr[0] := FALSE;
   S706_LM_DC_2ND_CLAMP6.Visu_Adv_Arr[1] := FALSE;
   S706_LM_DC_2ND_CLAMP6.Visu_Adv_Arr[2] := FALSE;
   S706_LM_DC_2ND_CLAMP6.Visu_Adv_Arr[3] := FALSE;
   S706_LM_DC_2ND_CLAMP6.Visu_Adv_Arr[4] := FALSE;
   S706_LM_DC_2ND_CLAMP6.Visu_Adv_Arr[5] := FALSE;
   S706_LM_DC_2ND_CLAMP6.Visu_Adv_Arr[6] := FALSE;
   S706_LM_DC_2ND_CLAMP6.Visu_Adv_Arr[7] := FALSE;
   S706_LM_DC_2ND_CLAMP6.Visu_Adv_Arr[8] := FALSE;
   S706_LM_DC_2ND_CLAMP6.Visu_Adv_Arr[9] := FALSE;
   S706_LM_DC_2ND_CLAMP6.Visu_Adv_Arr[10] := FALSE;
   S706_LM_DC_2ND_CLAMP6.Visu_Adv_Arr[11] := FALSE;
   S706_LM_DC_2ND_CLAMP6.Visu_Adv_Arr[12] := FALSE;
   S706_LM_DC_2ND_CLAMP6.Visu_Adv_Arr[13] := FALSE;
   S706_LM_DC_2ND_CLAMP6.Visu_Adv_Arr[14] := FALSE;
   S706_LM_DC_2ND_CLAMP6.Visu_Adv_Arr[15] := FALSE;
   S706_LM_DC_2ND_CLAMP6.Visu_Ret_Arr[0] := FALSE;
   S706_LM_DC_2ND_CLAMP6.Visu_Ret_Arr[1] := FALSE;
   S706_LM_DC_2ND_CLAMP6.Visu_Ret_Arr[2] := FALSE;
   S706_LM_DC_2ND_CLAMP6.Visu_Ret_Arr[3] := FALSE;
   S706_LM_DC_2ND_CLAMP6.Visu_Ret_Arr[4] := FALSE;
   S706_LM_DC_2ND_CLAMP6.Visu_Ret_Arr[5] := FALSE;
   S706_LM_DC_2ND_CLAMP6.Visu_Ret_Arr[6] := FALSE;
   S706_LM_DC_2ND_CLAMP6.Visu_Ret_Arr[7] := FALSE;
   S706_LM_DC_2ND_CLAMP6.Visu_Ret_Arr[8] := FALSE;
   S706_LM_DC_2ND_CLAMP6.Visu_Ret_Arr[9] := FALSE;
   S706_LM_DC_2ND_CLAMP6.Visu_Ret_Arr[10] := FALSE;
   S706_LM_DC_2ND_CLAMP6.Visu_Ret_Arr[11] := FALSE;
   S706_LM_DC_2ND_CLAMP6.Visu_Ret_Arr[12] := FALSE;
   S706_LM_DC_2ND_CLAMP6.Visu_Ret_Arr[13] := FALSE;
   S706_LM_DC_2ND_CLAMP6.Visu_Ret_Arr[14] := FALSE;
   S706_LM_DC_2ND_CLAMP6.Visu_Ret_Arr[15] := FALSE;
   S706_LM_DC_2ND_CLAMP6.BLK_Move_Ret := 0;
   S706_LM_DC_2ND_CLAMP6.Enable := FALSE;
   S706_LM_DC_2ND_CLAMP6.Adv_End := FALSE;
   S706_LM_DC_2ND_CLAMP6.Ret_End := FALSE;
   S706_LM_DC_2ND_CLAMP7.Enable_Aux := FALSE;
   S706_LM_DC_2ND_CLAMP7.Adv_Amount := 1;
   S706_LM_DC_2ND_CLAMP7.Ret_Amount := 1;
   S706_LM_DC_2ND_CLAMP7.LS_Adv1 := FALSE;
   S706_LM_DC_2ND_CLAMP7.LS_Ret1 := FALSE;
   S706_LM_DC_2ND_CLAMP7.LS_Adv2 := FALSE;
   S706_LM_DC_2ND_CLAMP7.LS_Ret2 := FALSE;
   S706_LM_DC_2ND_CLAMP7.LS_Adv3 := FALSE;
   S706_LM_DC_2ND_CLAMP7.LS_Ret3 := FALSE;
   S706_LM_DC_2ND_CLAMP7.LS_Adv4 := FALSE;
   S706_LM_DC_2ND_CLAMP7.LS_Ret4 := FALSE;
   S706_LM_DC_2ND_CLAMP7.SOL_Adv := FALSE;
   S706_LM_DC_2ND_CLAMP7.SOL_Ret := FALSE;
   S706_LM_DC_2ND_CLAMP7.M_Ready := TRUE;
   S706_LM_DC_2ND_CLAMP7.T_CHK1 := T#4S;
   S706_LM_DC_2ND_CLAMP7.T_CHK2 := T#4S;
   S706_LM_DC_2ND_CLAMP7.PB_Lamp_CHK := FALSE;
   S706_LM_DC_2ND_CLAMP7.PB_Error_Rst := FALSE;
   S706_LM_DC_2ND_CLAMP7.M_FLICK := FALSE;
   S706_LM_DC_2ND_CLAMP7.M_Adv_Err := FALSE;
   S706_LM_DC_2ND_CLAMP7.M_Ret_Err := FALSE;
   S706_LM_DC_2ND_CLAMP7.LP_Adv := FALSE;
   S706_LM_DC_2ND_CLAMP7.LP_Ret := FALSE;
   S706_LM_DC_2ND_CLAMP7.Visu_Adv := W#16#0;
   S706_LM_DC_2ND_CLAMP7.Visu_Ret := W#16#0;
   S706_LM_DC_2ND_CLAMP7.Error_T1.IN := FALSE;
   S706_LM_DC_2ND_CLAMP7.Error_T1.PT := T#4S;
   S706_LM_DC_2ND_CLAMP7.Error_T1.Q := FALSE;
   S706_LM_DC_2ND_CLAMP7.Error_T1.ET := T#0MS;
   S706_LM_DC_2ND_CLAMP7.Error_T1.STATE := B#16#0;
   S706_LM_DC_2ND_CLAMP7.Error_T1.STIME := T#0MS;
   S706_LM_DC_2ND_CLAMP7.Error_T1.ATIME := T#0MS;
   S706_LM_DC_2ND_CLAMP7.Error_T2.IN := FALSE;
   S706_LM_DC_2ND_CLAMP7.Error_T2.PT := T#4S;
   S706_LM_DC_2ND_CLAMP7.Error_T2.Q := FALSE;
   S706_LM_DC_2ND_CLAMP7.Error_T2.ET := T#0MS;
   S706_LM_DC_2ND_CLAMP7.Error_T2.STATE := B#16#0;
   S706_LM_DC_2ND_CLAMP7.Error_T2.STIME := T#0MS;
   S706_LM_DC_2ND_CLAMP7.Error_T2.ATIME := T#0MS;
   S706_LM_DC_2ND_CLAMP7.CHK_Aux1 := FALSE;
   S706_LM_DC_2ND_CLAMP7.CHK_Aux2 := FALSE;
   S706_LM_DC_2ND_CLAMP7.Error_T1_DN := FALSE;
   S706_LM_DC_2ND_CLAMP7.Error_T2_DN := FALSE;
   S706_LM_DC_2ND_CLAMP7.Adv_Memo := TRUE;
   S706_LM_DC_2ND_CLAMP7.Visu_Adv_Arr[0] := FALSE;
   S706_LM_DC_2ND_CLAMP7.Visu_Adv_Arr[1] := FALSE;
   S706_LM_DC_2ND_CLAMP7.Visu_Adv_Arr[2] := FALSE;
   S706_LM_DC_2ND_CLAMP7.Visu_Adv_Arr[3] := FALSE;
   S706_LM_DC_2ND_CLAMP7.Visu_Adv_Arr[4] := FALSE;
   S706_LM_DC_2ND_CLAMP7.Visu_Adv_Arr[5] := FALSE;
   S706_LM_DC_2ND_CLAMP7.Visu_Adv_Arr[6] := FALSE;
   S706_LM_DC_2ND_CLAMP7.Visu_Adv_Arr[7] := FALSE;
   S706_LM_DC_2ND_CLAMP7.Visu_Adv_Arr[8] := FALSE;
   S706_LM_DC_2ND_CLAMP7.Visu_Adv_Arr[9] := FALSE;
   S706_LM_DC_2ND_CLAMP7.Visu_Adv_Arr[10] := FALSE;
   S706_LM_DC_2ND_CLAMP7.Visu_Adv_Arr[11] := FALSE;
   S706_LM_DC_2ND_CLAMP7.Visu_Adv_Arr[12] := FALSE;
   S706_LM_DC_2ND_CLAMP7.Visu_Adv_Arr[13] := FALSE;
   S706_LM_DC_2ND_CLAMP7.Visu_Adv_Arr[14] := FALSE;
   S706_LM_DC_2ND_CLAMP7.Visu_Adv_Arr[15] := FALSE;
   S706_LM_DC_2ND_CLAMP7.Visu_Ret_Arr[0] := FALSE;
   S706_LM_DC_2ND_CLAMP7.Visu_Ret_Arr[1] := FALSE;
   S706_LM_DC_2ND_CLAMP7.Visu_Ret_Arr[2] := FALSE;
   S706_LM_DC_2ND_CLAMP7.Visu_Ret_Arr[3] := FALSE;
   S706_LM_DC_2ND_CLAMP7.Visu_Ret_Arr[4] := FALSE;
   S706_LM_DC_2ND_CLAMP7.Visu_Ret_Arr[5] := FALSE;
   S706_LM_DC_2ND_CLAMP7.Visu_Ret_Arr[6] := FALSE;
   S706_LM_DC_2ND_CLAMP7.Visu_Ret_Arr[7] := FALSE;
   S706_LM_DC_2ND_CLAMP7.Visu_Ret_Arr[8] := FALSE;
   S706_LM_DC_2ND_CLAMP7.Visu_Ret_Arr[9] := FALSE;
   S706_LM_DC_2ND_CLAMP7.Visu_Ret_Arr[10] := FALSE;
   S706_LM_DC_2ND_CLAMP7.Visu_Ret_Arr[11] := FALSE;
   S706_LM_DC_2ND_CLAMP7.Visu_Ret_Arr[12] := FALSE;
   S706_LM_DC_2ND_CLAMP7.Visu_Ret_Arr[13] := FALSE;
   S706_LM_DC_2ND_CLAMP7.Visu_Ret_Arr[14] := FALSE;
   S706_LM_DC_2ND_CLAMP7.Visu_Ret_Arr[15] := FALSE;
   S706_LM_DC_2ND_CLAMP7.BLK_Move_Ret := 0;
   S706_LM_DC_2ND_CLAMP7.Enable := FALSE;
   S706_LM_DC_2ND_CLAMP7.Adv_End := FALSE;
   S706_LM_DC_2ND_CLAMP7.Ret_End := FALSE;
   S706_LM_DC_1ST_CLAMP5.Enable_Aux := FALSE;
   S706_LM_DC_1ST_CLAMP5.Adv_Amount := 1;
   S706_LM_DC_1ST_CLAMP5.Ret_Amount := 1;
   S706_LM_DC_1ST_CLAMP5.LS_Adv1 := FALSE;
   S706_LM_DC_1ST_CLAMP5.LS_Ret1 := FALSE;
   S706_LM_DC_1ST_CLAMP5.LS_Adv2 := FALSE;
   S706_LM_DC_1ST_CLAMP5.LS_Ret2 := FALSE;
   S706_LM_DC_1ST_CLAMP5.LS_Adv3 := FALSE;
   S706_LM_DC_1ST_CLAMP5.LS_Ret3 := FALSE;
   S706_LM_DC_1ST_CLAMP5.LS_Adv4 := FALSE;
   S706_LM_DC_1ST_CLAMP5.LS_Ret4 := FALSE;
   S706_LM_DC_1ST_CLAMP5.SOL_Adv := FALSE;
   S706_LM_DC_1ST_CLAMP5.SOL_Ret := FALSE;
   S706_LM_DC_1ST_CLAMP5.M_Ready := TRUE;
   S706_LM_DC_1ST_CLAMP5.T_CHK1 := T#4S;
   S706_LM_DC_1ST_CLAMP5.T_CHK2 := T#4S;
   S706_LM_DC_1ST_CLAMP5.PB_Lamp_CHK := FALSE;
   S706_LM_DC_1ST_CLAMP5.PB_Error_Rst := FALSE;
   S706_LM_DC_1ST_CLAMP5.M_FLICK := FALSE;
   S706_LM_DC_1ST_CLAMP5.M_Adv_Err := FALSE;
   S706_LM_DC_1ST_CLAMP5.M_Ret_Err := FALSE;
   S706_LM_DC_1ST_CLAMP5.LP_Adv := FALSE;
   S706_LM_DC_1ST_CLAMP5.LP_Ret := FALSE;
   S706_LM_DC_1ST_CLAMP5.Visu_Adv := W#16#0;
   S706_LM_DC_1ST_CLAMP5.Visu_Ret := W#16#0;
   S706_LM_DC_1ST_CLAMP5.Error_T1.IN := FALSE;
   S706_LM_DC_1ST_CLAMP5.Error_T1.PT := T#4S;
   S706_LM_DC_1ST_CLAMP5.Error_T1.Q := FALSE;
   S706_LM_DC_1ST_CLAMP5.Error_T1.ET := T#0MS;
   S706_LM_DC_1ST_CLAMP5.Error_T1.STATE := B#16#0;
   S706_LM_DC_1ST_CLAMP5.Error_T1.STIME := T#0MS;
   S706_LM_DC_1ST_CLAMP5.Error_T1.ATIME := T#0MS;
   S706_LM_DC_1ST_CLAMP5.Error_T2.IN := FALSE;
   S706_LM_DC_1ST_CLAMP5.Error_T2.PT := T#4S;
   S706_LM_DC_1ST_CLAMP5.Error_T2.Q := FALSE;
   S706_LM_DC_1ST_CLAMP5.Error_T2.ET := T#0MS;
   S706_LM_DC_1ST_CLAMP5.Error_T2.STATE := B#16#0;
   S706_LM_DC_1ST_CLAMP5.Error_T2.STIME := T#0MS;
   S706_LM_DC_1ST_CLAMP5.Error_T2.ATIME := T#0MS;
   S706_LM_DC_1ST_CLAMP5.CHK_Aux1 := FALSE;
   S706_LM_DC_1ST_CLAMP5.CHK_Aux2 := FALSE;
   S706_LM_DC_1ST_CLAMP5.Error_T1_DN := FALSE;
   S706_LM_DC_1ST_CLAMP5.Error_T2_DN := FALSE;
   S706_LM_DC_1ST_CLAMP5.Adv_Memo := TRUE;
   S706_LM_DC_1ST_CLAMP5.Visu_Adv_Arr[0] := FALSE;
   S706_LM_DC_1ST_CLAMP5.Visu_Adv_Arr[1] := FALSE;
   S706_LM_DC_1ST_CLAMP5.Visu_Adv_Arr[2] := FALSE;
   S706_LM_DC_1ST_CLAMP5.Visu_Adv_Arr[3] := FALSE;
   S706_LM_DC_1ST_CLAMP5.Visu_Adv_Arr[4] := FALSE;
   S706_LM_DC_1ST_CLAMP5.Visu_Adv_Arr[5] := FALSE;
   S706_LM_DC_1ST_CLAMP5.Visu_Adv_Arr[6] := FALSE;
   S706_LM_DC_1ST_CLAMP5.Visu_Adv_Arr[7] := FALSE;
   S706_LM_DC_1ST_CLAMP5.Visu_Adv_Arr[8] := FALSE;
   S706_LM_DC_1ST_CLAMP5.Visu_Adv_Arr[9] := FALSE;
   S706_LM_DC_1ST_CLAMP5.Visu_Adv_Arr[10] := FALSE;
   S706_LM_DC_1ST_CLAMP5.Visu_Adv_Arr[11] := FALSE;
   S706_LM_DC_1ST_CLAMP5.Visu_Adv_Arr[12] := FALSE;
   S706_LM_DC_1ST_CLAMP5.Visu_Adv_Arr[13] := FALSE;
   S706_LM_DC_1ST_CLAMP5.Visu_Adv_Arr[14] := FALSE;
   S706_LM_DC_1ST_CLAMP5.Visu_Adv_Arr[15] := FALSE;
   S706_LM_DC_1ST_CLAMP5.Visu_Ret_Arr[0] := FALSE;
   S706_LM_DC_1ST_CLAMP5.Visu_Ret_Arr[1] := FALSE;
   S706_LM_DC_1ST_CLAMP5.Visu_Ret_Arr[2] := FALSE;
   S706_LM_DC_1ST_CLAMP5.Visu_Ret_Arr[3] := FALSE;
   S706_LM_DC_1ST_CLAMP5.Visu_Ret_Arr[4] := FALSE;
   S706_LM_DC_1ST_CLAMP5.Visu_Ret_Arr[5] := FALSE;
   S706_LM_DC_1ST_CLAMP5.Visu_Ret_Arr[6] := FALSE;
   S706_LM_DC_1ST_CLAMP5.Visu_Ret_Arr[7] := FALSE;
   S706_LM_DC_1ST_CLAMP5.Visu_Ret_Arr[8] := FALSE;
   S706_LM_DC_1ST_CLAMP5.Visu_Ret_Arr[9] := FALSE;
   S706_LM_DC_1ST_CLAMP5.Visu_Ret_Arr[10] := FALSE;
   S706_LM_DC_1ST_CLAMP5.Visu_Ret_Arr[11] := FALSE;
   S706_LM_DC_1ST_CLAMP5.Visu_Ret_Arr[12] := FALSE;
   S706_LM_DC_1ST_CLAMP5.Visu_Ret_Arr[13] := FALSE;
   S706_LM_DC_1ST_CLAMP5.Visu_Ret_Arr[14] := FALSE;
   S706_LM_DC_1ST_CLAMP5.Visu_Ret_Arr[15] := FALSE;
   S706_LM_DC_1ST_CLAMP5.BLK_Move_Ret := 0;
   S706_LM_DC_1ST_CLAMP5.Enable := FALSE;
   S706_LM_DC_1ST_CLAMP5.Adv_End := FALSE;
   S706_LM_DC_1ST_CLAMP5.Ret_End := FALSE;
END_DATA_BLOCK

FUNCTION FC 123 : VOID
TITLE =
NAME : DAECHA
VERSION : 0.1

BEGIN
NETWORK
TITLE =
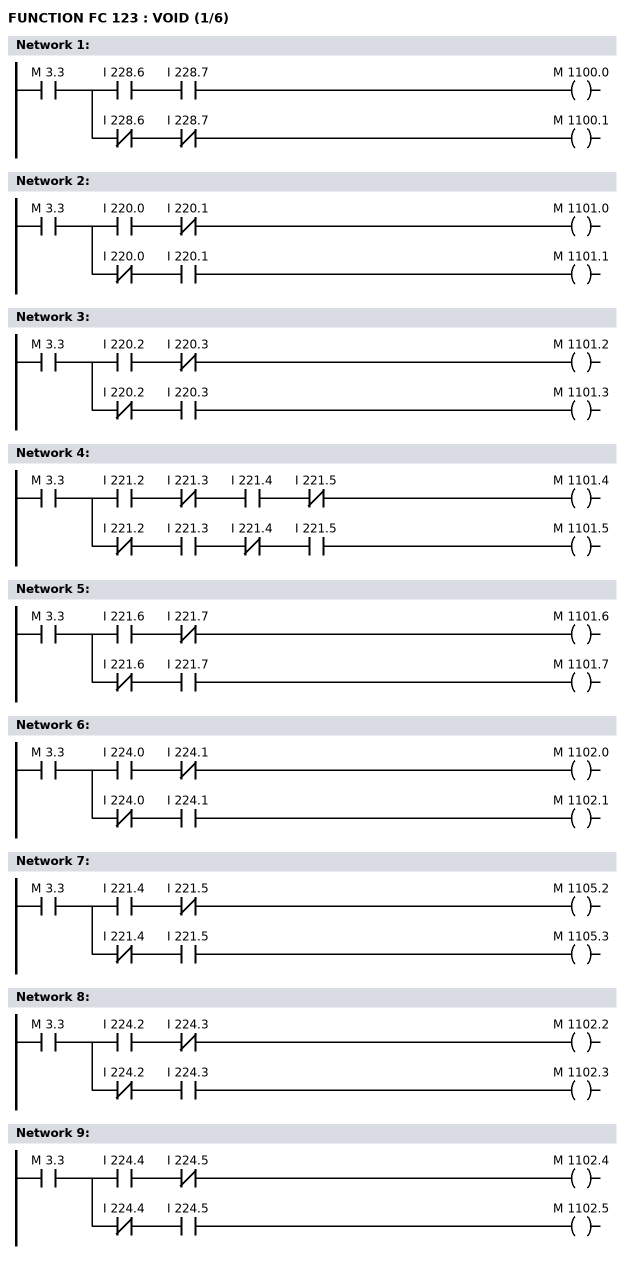

      A     M      3.3;
      =     L      0.0;
      A     L      0.0;
      A     I    228.6;
      A     I    228.7;
      =     M   1100.0;
      A     L      0.0;
      AN    I    228.6;
      AN    I    228.7;
      =     M   1100.1;
NETWORK
TITLE =

      A     M      3.3;
      =     L      0.0;
      A     L      0.0;
      A     I    220.0;
      AN    I    220.1;
      =     M   1101.0;
      A     L      0.0;
      AN    I    220.0;
      A     I    220.1;
      =     M   1101.1;
NETWORK
TITLE =

